# B&R Automation Studio project MIG1 (part 9)

### WSI_lib.c
```c
/********************************************************************
 * COPYRIGHT --
 ********************************************************************
 * Package: Lib
 * File: WSI_lib.c
 * Author: ckaczkowski
 * Created: June 18, 2014
 *******************************************************************/

#include <bur/plctypes.h>
#ifdef _DEFAULT_INCLUDES
	#include <AsDefault.h>
#endif

#ifndef _WSITYPES_C
#define _WSITYPES_C

//#define NULL 0

/* Prototyping of functions and function blocks */

float Scal(float x, AzzScal_typ* scale);
float LimScal(float x, AzzLimScal_typ* scale);

DINT Errors(ERROR_Mgr_typ *mgr , char type , unsigned short indx , unsigned long val);

DINT AckAllErrors(ERROR_Mgr_typ *mgr);

DINT StateVectorSrv(StateVectorProxy_typ *vect , UINT thread);

UINT Bool2Uint(plcbit in);
plcbit Uint2Bool(UINT in);

char* UDINT2ASC(UDINT val);
UDINT ASC2UDINT(char *p);

INT ABS_INT(INT x);

float getFromCalib(float x , Calib_Param_typ* calib , UINT type);

static UDINT hash_of_binary_array(char *key, int len);

///////////////////////////////////////////////////////
//////   Functions from Paul
void AzzLinSpline(AzzLinSpline_typ *lcr);
void AzzSlimPID(AzzSlimPID_typ *lcr);
void AzzRamp(AzzRamp_typ *lcr);
void AzzMovAvgFlt(AzzMovAvgFlt_typ *lcr) ;
void AzzLimScal(AzzLimScal_typ *lcr);
void AzzScal(AzzScal_typ *lcr);
void AzzTON(AzzTON_typ *t);
void HCRSPFazz(HCRSPFazz_type* inst);

void AzzLinSpline(AzzLinSpline_typ *lcr){
UINT outer , inner;
INT i;
float tempX, tempY;
float slope , delta;

	if(!lcr->pNodeVec)
		return;

	if(lcr->NbNodes < 2)
		return;

	//////////////////////////////////////////////

	if(lcr->Invert){

		if(lcr->x < lcr->pNodeVec[0].Y)
			lcr->y = lcr->pNodeVec[0].X;
		else if(lcr->x > lcr->pNodeVec[lcr->NbNodes-1].Y)
			lcr->y = lcr->pNodeVec[lcr->NbNodes-1].X;

		else{

			i = lcr->NbNodes-2;
			while((lcr->x < lcr->pNodeVec[i].Y) && (i > 0) ) { i--; }

			lcr->_i = i;

			delta = lcr->pNodeVec[i+1].Y - lcr->pNodeVec[i].Y;

			if(delta != 0.0)
				slope = (lcr->pNodeVec[i+1].X - lcr->pNodeVec[i].X)/delta;
			else
				slope =0;

			lcr->y = lcr->pNodeVec[i].X + slope * (lcr->x - lcr->pNodeVec[i].Y);

		}

	}
	else{

		if(lcr->x < lcr->pNodeVec[0].X)
			lcr->y = lcr->pNodeVec[0].Y;
		else if(lcr->x > lcr->pNodeVec[lcr->NbNodes-1].X)
			lcr->y = lcr->pNodeVec[lcr->NbNodes-1].Y;

		else{

			i = lcr->NbNodes-2;
			while((lcr->x < lcr->pNodeVec[i].X) && (i > 0) ) { i--; }

			lcr->_i = i;

			delta = lcr->pNodeVec[i+1].X - lcr->pNodeVec[i].X;

			if(delta != 0.0)
				slope = (lcr->pNodeVec[i+1].Y - lcr->pNodeVec[i].Y)/delta;
			else
				slope =0;

			lcr->y = lcr->pNodeVec[i].Y + slope * (lcr->x - lcr->pNodeVec[i].X);

		}

	}

	///////////////////////////////////////////////
	if(lcr->Update){
		lcr->Update = 0;

		//Bubble sort
		 for(outer=0;outer<lcr->NbNodes-1;outer++)
		 {
			 for(inner=outer+1;inner<lcr->NbNodes;inner++)
			 {

			 	if(lcr->Invert){

					 if(lcr->pNodeVec[outer].Y > lcr->pNodeVec[inner].Y)
					 {
						 tempX=lcr->pNodeVec[outer].X;
						 tempY=lcr->pNodeVec[outer].Y;

						 lcr->pNodeVec[outer].X = lcr->pNodeVec[inner].X;
						 lcr->pNodeVec[outer].Y = lcr->pNodeVec[inner].Y;

						 lcr->pNodeVec[inner].X = tempX;
						 lcr->pNodeVec[inner].Y = tempX;

					 }

			 	}
				else{

					if(lcr->pNodeVec[outer].X > lcr->pNodeVec[inner].X)
					 {
						 tempX=lcr->pNodeVec[outer].X;
						 tempY=lcr->pNodeVec[outer].Y;

						 lcr->pNodeVec[outer].X = lcr->pNodeVec[inner].X;
						 lcr->pNodeVec[outer].Y = lcr->pNodeVec[inner].Y;

						 lcr->pNodeVec[inner].X = tempX;
						 lcr->pNodeVec[inner].Y = tempX;

					 }

				}
			 }
		 }

	}

}

void AzzTON(AzzTON_typ *t) {
  if (t->IN) {
    // Check for rising edge
    if (!t->M) {
      t->StartTime = clock_ms();
    }

    // Determine elapsed time
    t->ET = clock_ms() - t->StartTime;

    // Check if the elapsed time has reached delay time
    if (t->ET >= t->PT) {
      t->Q = 1;
      t->ET = t->PT;
    } else {
      t->Q = 0;
    }

  } else {
    t->Q = 0;
    t->ET = 0;
  }

  // Set M to IN to allow checking for rising edge
  t->M = t->IN;
}

void AzzRamp(AzzRamp_typ *lcr) {
float x = lcr->x, y = lcr->y_old;
float dt;
DINT time , deltaT;

	lcr->status = 0;

	if ( !lcr->enable ) {

		lcr->timestore1 = AsIOTimeStamp();
		lcr->status = 65534;
		return;

	}

	// Check parameters
	  // rate up and rate down have to be greater than zero
	if ( lcr->dy_up <= 0 || lcr->dy_down <= 0 ) {
	  lcr->status = 12034;
	  return;
	}

	if ( lcr->set ) { // Set default value

		lcr->set = 0;

		y = lcr->y_set;

		lcr->y_old = y;

		lcr->y = y;

		lcr->timestore1 = AsIOTimeStamp();

	}
	else {
		// Process Ramp

		time = AsIOTimeStamp();
		deltaT = (time- lcr->timestore1);
		lcr->timestore1 = time;

		if(deltaT > 0 && (deltaT < 0x4FFFFFFF))
			dt = (float)(deltaT) / 1000000.0;
		else
			dt = 0.0;

		lcr->dt = dt;

		/*
		// Calculate new value
		if ( x > y && y > 0 ) {
			y = lcr->y_old + ( dt * lcr->dy_up );
			if(y > x)
				y = x;

		} else if ( x < y && y < 0 ) {
			y = lcr->y_old - ( dt * lcr->dy_up );
			if(y < x)
				y = x;

		} else if ( x < y && y > 0 ) {
			y = lcr->y_old - ( dt * lcr->dy_down );
			if(y < x)
				y = x;

		} else if ( x > y && y < 0 ) {
			y = lcr->y_old + ( dt * lcr->dy_down );
			if(y > x)
				y = x;
		}
		*/

		if ( x > y ) {
			y = lcr->y_old + ( dt * lcr->dy_up );
			if(y > x)
				y = x;

		} else if ( x < y ) {
			y = lcr->y_old - ( dt * lcr->dy_down );
			if(y < x)
				y = x;
		}

		// Check limits
		if (y >= lcr->y_max ) {
		  y = lcr->y_max;
		  lcr->max_limit = 1;

		}

		else if(y <= lcr->y_min ) {
		  y = lcr->y_min;
		  lcr->min_limit = 1;

		}

		lcr->y = y;

		lcr->x_reached = (lcr->y == lcr->x)? 1:0;
		lcr->y_old = y;

	}

}

void AzzMovAvgFlt(AzzMovAvgFlt_typ *lcr) {

  float *ptr;
  double *sum = (double*)&lcr->sum_old;
  int i;

  //lcr->y = lcr->x ;
  //return;

  if(!lcr){
  	lcr->status = -1;
	return;
  }

  if(lcr->base == 0){
  	lcr->status = -2;
	return;
  }

  lcr->status = 0;

  if ( lcr->enable ) {
    // Default to successful status
    lcr->status = 0;

    // If base has changed, re-allocate buffer
    if ( lcr->base != lcr->base_old || ( (void *)lcr->p_xold == 0 ) ) {

      // Free the old buffer
	 if((lcr->p_xold != 0 ) && lcr->base_old > 0){
		  if(TMP_free(lcr->base_old , (void**) lcr->p_xold)){
		  	return;
		  }
		  else
		  	lcr->base_old = 0;

	 }
	 else{ // Memory leack

	 	 lcr->base_old = 0;
		 lcr->p_xold = 0;

	 }

      //if ( (void *)lcr->p_xold != 0 )
        //free((void *)lcr->p_xold);

      // Allocate new buffer
      //lcr->p_xold = (unsigned long)malloc(lcr->base * sizeof(lcr->x));
      if(TMP_alloc(lcr->base * sizeof(float)  , (void**)&lcr->p_xold))
	  	return;
	  else
		lcr->base_old = lcr->base;

      ptr = (float*)lcr->p_xold;

      // Set buffer to initial values (current x)
      if (ptr != 0) {
        // Loop through whole buffer
        for( i = 0; i < lcr->base; i++ ) {
          *ptr = lcr->x;
          ptr++;
        }
      } else {
        lcr->status = 12018;
        return;
      }

      // Set sum
      *sum = lcr->x * lcr->base;

	  lcr->y = (*sum) / lcr->base;

      // Set index
      lcr->i_xold = 0;
    }

	 //return;
	if ( lcr->i_xold >= lcr->base )
      lcr->i_xold = 0;

	ptr = (float*)lcr->p_xold;
    // Calculate new sum
    *sum = *sum - *(ptr + lcr->i_xold) + lcr->x;

    // Replace x value in buffer
    *(ptr + lcr->i_xold) = lcr->x;

    // Increase index and ring around the buffer if necessary
    lcr->i_xold ++;

    // Calculate new avg
    lcr->y = (*sum) / lcr->base;

  }

  else {

    lcr->status = 65534;
  }

}

void AzzSlimPID(AzzSlimPID_typ *lcr) {

  AzzPID_typ *pid = &lcr->PID_inst;
  azzslimpid_par_typ *para = lcr->pPar;
  float p, i, d, error, dt;
  DINT time , deltaT;

  // TODO - Ensure that the derivative term does not go crazy first scan
  // We are not using the derivative

  if (lcr->enable) {
	    // Get current time
	    time = AsIOTimeStamp();

	    // Determine error
	      // Includes feedback damping
	      // e_fbk = Kfbk / Kp * (Ytotal - Y)

	    //error = lcr->W - lcr->X - pid->e_fbk;
	    error = lcr->W - lcr->X ;

		deltaT = (time - pid->last_time);

		if(deltaT > 0 && (deltaT < 0x4FFFFFFF))
	    	dt = (float)(deltaT) / 1000000.0;
		else
			dt = 0.0;

		lcr->dt = dt;
		lcr->e = error;

	    // Proportional control
	    p = para->Kp * error;

	    // Integral control
	    //pid->i_sum += error * dt;
	    pid->i_sum += ((error - pid->e_fbk) * para->Kp * dt);

		if(para->Tn > 0)
	    	i = pid->i_sum / para->Tn;
		else
			i = 0;

	    // Derivative control
	    if(dt > 0)
	    	d = ((lcr->X - pid->d_old) / dt) * para->Tv * para->Kp ;
		else
			d = 0.0;

	    pid->d_old = lcr->X;

	    // Set output variable
	    lcr->Y = p + i + d;

	    // Limit output variable
	    if (lcr->Y > para->Y_max) {
	      pid->e_fbk = para->Kfbk * (lcr->Y - para->Y_max);
	      lcr->Y = para->Y_max;
	    } else if (lcr->Y < para->Y_min) {
	      pid->e_fbk = para->Kfbk * (lcr->Y - para->Y_min);
	      lcr->Y = para->Y_min;
	    } else {
	      pid->e_fbk = 0;
	    }

  } else {

  	i = pid->i_sum = 0;
    lcr->status = 65534;
  }

  pid->last_time = AsIOTimeStamp();

}

void AzzScal(AzzScal_typ *lcr) {
  REAL k, d;

  if (lcr->x1 != lcr->x2) {
    k = (lcr->y2 - lcr->y1) / (lcr->x2 - lcr->x1);
    lcr->y = lcr->y1 + (k * (lcr->x - lcr->x1));

  } else {
    lcr->y = 0;
  }

}

void AzzLimScal(AzzLimScal_typ *lcr) {
  REAL *high, *low;

  // Run LCRScal - this function is the same except for limits
  AzzScal((AzzScal_typ *)lcr);

  // Find high limit and low limit
  if (lcr->y1 < lcr->y2) {
    high = &lcr->y2;
    low = &lcr->y1;
  } else {
    low = &lcr->y2;
    high = &lcr->y1;
  }

  // Limit y to be between the high and low values
  if (lcr->y > *high)
    lcr->y = *high;
  if (lcr->y < *low)
    lcr->y = *low;

}

//////////    END of New Functions /////////////////////
/////////////////////////////////////////////////////

float LimScal(float x, AzzLimScal_typ* scale){

	scale->x = x;
	AzzLimScal(scale);

	return scale->y;
}

float Scal(float x, AzzScal_typ* scale){

	scale->x = x;
	AzzScal(scale);

	return scale->y;
}

DINT Errors(ERROR_Mgr_typ *mgr , char type , unsigned short indx , unsigned long val){

	if(!mgr->logs[indx].status){

		mgr->lastItemIndx++;
		if(mgr->lastItemIndx >= 64)
			mgr->lastItemIndx = 0;

		mgr->logs[indx].status = 1;
		mgr->logs[indx].value = val;
		mgr->history[mgr->lastItemIndx] = indx;

		if(type > 0){
			if(type >= mgr->Error) // set only higher priority error
				mgr->Error = type;
		}
		else
			mgr->Error = type;

		return 1;

	}
	else
		return 0;
}

DINT AckAllErrors(ERROR_Mgr_typ *mgr){
	int i;

	// Never clear fatal error
	if (mgr->Error < 0)
		return -1;

	for( i = 0 ; i < 64 ; i++){

		mgr->logs[i].status = 0;

		mgr->history[i] = 0;

	}

	mgr->Error = 0;
	mgr->lastItemIndx = 0;

	return 1;

}

DINT StateVectorSrv(StateVectorProxy_typ *vect , UINT thread){

	if(vect->testMode)
		return;

	/*****************************************/
	///    VECTOR  SERVER

	if(!vect->simul){

		vect->OutVect.Mode = vect->Mode ;

		switch(vect->Mode){

			case vectSt_Mode_Idle:

				vect->OutVect.volt = 0.0;
				vect->OutVect.vel = 0.0;

				break;

			case vectSt_Mode_Hold:

				break;

			case vectSt_Mode_Home:

				break;

			case vectSt_Mode_Pos:

				vect->OutVect.volt = 0.0;
				vect->OutVect.amp  = 0.0;

				//if(thread == vect->Indx )
					vect->OutVect.x = vect->InVal;

				break;

			case vectSt_Mode_Vel:

				vect->OutVect.volt = 0.0;
				vect->OutVect.amp  = 0.0;

				//if(thread == vect->Indx )
					vect->OutVect.vel = vect->InVal;

				break;

			case vectSt_Mode_Volt:

				vect->OutVect.amp  = 0.0;

				//if(thread == vect->Indx )
					vect->OutVect.volt = vect->InVal;

				vect->OutVect.vel = 0;

				break;

			case vectSt_Mode_Torq:

				vect->OutVect.volt = 0.0;

				//if(thread == vect->Indx )
					vect->OutVect.amp = vect->InVal;

				vect->OutVect.vel = 0;

				break;

			case vectSt_Mode_PT:

				vect->OutVect.volt = 0.0;
				vect->OutVect.amp  = 0.0;
				vect->OutVect.x = vect->InVal;

				break;

		}
	}
	else{

		vect->FbkVect.Mode = vect->Mode;

		switch(vect->Mode){

			case vectSt_Mode_Idle:

				vect->FbkVect.x = 0;
				vect->FbkVect.vel = 0;

				break;

			case vectSt_Mode_Hold:

				break;

			case vectSt_Mode_Home:

				break;

			case vectSt_Mode_Pos:

				vect->FbkVect.x = vect->InVal;

				break;

			case vectSt_Mode_Vel:

				vect->FbkVect.vel = vect->InVal;

				break;

			case vectSt_Mode_Volt:

				vect->FbkVect.volt = vect->InVal;

				break;

			case vectSt_Mode_Torq:

				vect->FbkVect.amp = vect->InVal;

				break;

			case vectSt_Mode_PT:

				vect->FbkVect.x = vect->InVal;
				//vect->OutVect.x = vect->InVal;

				break;

		}

	}

	return 1;

}

UINT Bool2Uint(plcbit in){

	if(in)
		return 1;
	else
		return 0;

}

plcbit Uint2Bool(UINT in){

	if(in > 0)
		return 1;
	else
		return 0;

}

char* UDINT2ASC(UDINT val){
static char ret[5];
UDINT mask;
int i;

	mask = 0x000000FF;

	for(i=3 ; i >= 0 ; i--){

		ret[i] = (char)(val & mask);
		val = val >> 8;

	}
	ret[4] = 0;
	return ret;

}

UDINT ASC2UDINT(char *p){
UDINT val;
int i;

	val = 0;

	for(i=0 ; i < 4  ; i++){
		val = val<<8;
		val += p[i];
	}

	return val;

}
INT ABS_INT(INT x){

	if( x >= 0)
		return x;
	else
		return x*(-1);

}

float getFromCalib(float x , Calib_Param_typ* calib , UINT type){
float ret; float _x;
AzzScal_typ scale;

	if(!calib)
		return 0.0;

	if(x == 0.0)
		return 0.0;

	if(x < 0.0)
		_x = x * (-1.0);
	else
		_x = x;

	switch(type){

		case CALIB_ONE2ONE:

			ret = _x;

		break;

		case CALIB_2POINTS:

			scale.x = _x;
			scale.x1 = calib->val[0];
			scale.y1 = calib->val[1];
			scale.x2 = calib->val[2];
			scale.y2 = calib->val[3];

			if( _x < scale.x1)
				ret = (_x/scale.x1) * scale.y1;

			else {
				AzzScal(&scale);
				ret = scale.y;
			}

		break;

		case CALIB_2POINTS_4OFF:

			scale.x = _x;
			scale.x1 = calib->val[4];
			scale.y1 = calib->val[5];
			scale.x2 = calib->val[6];
			scale.y2 = calib->val[7];

			if( _x < scale.x1)
				ret = (_x/scale.x1) * scale.y1;

			else {
				AzzScal(&scale);
				ret = scale.y;
			}

		break;

		case CALIB_2POINTS_INV:

			scale.x = _x;
			scale.x1 = calib->val[1];
			scale.y1 = calib->val[0];
			scale.x2 = calib->val[3];
			scale.y2 = calib->val[2];

			if( _x < scale.x1)
				ret = (_x/scale.x1) * scale.y1;

			else {
				AzzScal(&scale);
				ret = scale.y;
			}

		break;

		case CALIB_2POINTS_4OFF_INV:

			scale.x = _x;
			scale.x1 = calib->val[5];
			scale.y1 = calib->val[4];
			scale.x2 = calib->val[7];
			scale.y2 = calib->val[6];

			if( _x < scale.x1)
				ret = (_x/scale.x1) * scale.y1;

			else {

				AzzScal(&scale);
				ret = scale.y;
			}

		break;

	}

	// Symetric to zero
	if(x <  0.0)
		ret = ret * (-1.);

	return ret;

}

static UDINT hash_of_binary_array(char *key, int len)
{
	unsigned int hash, i;
	for(hash = i = 0; i < len; ++i)
	{
		hash += key[i];
		hash += (hash << 10);
		hash ^= (hash >> 6);
	}
	hash += (hash << 3);
	hash ^= (hash >> 11);
	hash += (hash << 15);
	return hash;
}

///   New Path Generator created March 2019 by CK
void HCRSPFazz(HCRSPFazz_type* inst){
float dist, a , d , v , v02 , ad2 , x , s ;
float S_end , S_in , V_in , V0 , V_max;
float dir;
UINT t;
float deltaT;

	if(!inst)
		return;
/*****************************************/

	if(!inst->Intr._Set_home && inst->Set_home){
		// This is new for conveniance
		inst->Set_home = 0;

		inst->s_set = inst->s_home;
		inst->v_set = 0;
		inst->a_set = 0;

		inst->Intr.step = 0;

	}

	if(!inst->Intr._Stop && inst->Stop){

		// This is new for conveniance
		inst->Stop = 0;

		inst->v_set = 0;
		inst->a_set = 0;

		inst->Intr.step = 0;

	}

	if(!inst->Intr._Brake && inst->Brake){

		d = (inst->v_set > 0)? inst->pMove_Para->aDec_pos : inst->pMove_Para->aDec_neg;
		dir = (inst->v_set > 0.0)? 1.0:-1.0;

		/*
		inst->s_end = ((inst->v_set * inst->v_set )/d/2.0)*dir + inst->s_set;

		inst->Intr.step = 1;
		*/

		inst->Intr.S0 = ((inst->v_set * inst->v_set )/d/2.0)*dir;
		inst->Intr.segm[0].s = inst->Intr.S0  + inst->s_set ;
		inst->Intr.segm[0].v = 0;
		inst->Intr.segm[0].a = -d * dir;

		inst->Intr.S1 = 0.0;
		inst->Intr.segm[1].s = inst->Intr.segm[0].s;
		inst->Intr.segm[1].v = 0;
		inst->Intr.segm[1].a = 0;

		inst->Intr.S2 = 0.0;
		inst->Intr.segm[2].s = inst->Intr.segm[0].s;
		inst->Intr.segm[2].v = 0;
		inst->Intr.segm[2].a = 0;

		inst->Intr.S3 = 0.0;
		inst->Intr.segm[3].s = inst->Intr.segm[0].s;
		inst->Intr.segm[3].v = 0;
		inst->Intr.segm[3].a = 0;

		inst->Intr.indx = 0;
		inst->elapseTime = 0.0;
		inst->Reached = 0;
		inst->Intr.step = 3;

	}

	if(!inst->Intr._Init && inst->Init )
		inst->Intr.step = 1;

	switch(inst->Intr.step){

		//// Verify if current velocity in bigger then maximum velocity
		case 1:

			strcpy(inst->Intr.statusTxt , "");

			inst->Reached = 0;

			inst->Intr.segm[0].s = inst->s_set;
			inst->Intr.segm[0].v = inst->v_set;
			inst->Intr.segm[0].a = 0.0;

			inst->Intr.S0 = 0;
			////////////////////////////////////////////////////////////////////////////////////////
			// Check if movement direction change is necessary

			dist = inst->s_end - inst->Intr.segm[0].s;
			d = (inst->Intr.segm[0].v > 0)? inst->pMove_Para->aDec_pos : inst->pMove_Para->aDec_neg;

			s = ((inst->v_set * inst->v_set)/d)/2.0;

			if((fabsf(dist) < s) 					// Distance is smaller then coming from deceleration
				|| ((dist *  inst->v_set)<0.0)){ 	// Running in oposite direction

				strcpy(inst->Intr.statusTxt , "Change move direction");

				if(inst->Intr.segm[0].v > 0){

					inst->Intr.S0 = s;
					inst->Intr.segm[0].s += s;
					inst->Intr.segm[0].v = 0.0;
					inst->Intr.segm[0].a = -d;

				}
				if(inst->Intr.segm[0].v < 0){

					inst->Intr.S0 = -s;
					inst->Intr.segm[0].s -= s;
					inst->Intr.segm[0].v = 0.0;
					inst->Intr.segm[0].a = d;

				}

				goto CALCULATE_TRAPEZOID;

			}

			///////////////////////////////////////////////////////////////////////////////////////////
			///  Check Speed above maximum

			if(inst->v_set > 0.0)
				V_max = inst->pMove_Para->vC_pos;
			else if(inst->v_set < 0.0)
				V_max = inst->pMove_Para->vC_neg;

			if(fabsf(inst->v_set) > V_max){ // reduce speed first{

				if(inst->v_set > 0.0){

					inst->Intr.segm[0].v = V_max;
					inst->Intr.segm[0].a = -inst->pMove_Para->aDec_pos;

					x = (fabsf(inst->v_set) - V_max );
					inst->Intr.S0 = (x * x)/ inst->pMove_Para->aDec_pos /2.0 ;
					inst->Intr.S0 += inst->Intr.segm[0].v * x/inst->pMove_Para->aDec_pos;

					inst->Intr.segm[0].s += inst->Intr.S0;

					strcpy(inst->Intr.statusTxt , "Max Pos Vel");
				}
				else if(inst->v_set < 0.0){

					inst->Intr.segm[0].v = -V_max;
					inst->Intr.segm[0].a = inst->pMove_Para->aDec_neg;

					x = (fabsf(inst->v_set) - V_max );
					inst->Intr.S0 = (x * x)/ inst->pMove_Para->aDec_neg /(-2.0) ;
					inst->Intr.S0 += inst->Intr.segm[0].v * x/inst->pMove_Para->aDec_neg;

					inst->Intr.segm[0].s += inst->Intr.S0;

					strcpy(inst->Intr.statusTxt , "Max Neg Vel");
				}

			}

			CALCULATE_TRAPEZOID:
			//////////////////////////////////////////////////////////
			///  Calculate Segments 1 , 2 , 3
			S_end = inst->s_end;
			S_in  = inst->Intr.segm[0].s ;
			V_in  = inst->Intr.segm[0].v ;

			dir = (S_end > S_in)? 1.0:-1.0;

			if(dir > 0){
				a = inst->pMove_Para->aAcc_pos;
				d = inst->pMove_Para->aDec_pos;
			}
			else if(dir < 0){

				a = inst->pMove_Para->aAcc_neg;
				d = inst->pMove_Para->aDec_neg;
			}
			else{

				strcpy(inst->Intr.statusTxt , "No Trapezoid");

			}

			inst->Intr.segm[1].a = a ;
			inst->Intr.segm[2].a = 0;
			inst->Intr.segm[3].a = -d  ;

			////////////////////////////////////////////
			// Calculate maximum velocity

			dist = fabsf(S_end - S_in);
			V0 = fabsf(V_in);

			v02 = (V0 * V0)/ (2.0 * a);
			ad2 = (1.0/(2*a)) + (1.0/(2*d));

			 v = (dist + v02)/ad2;

			 v = sqrtf(v);

			////////////////////////

			if(dir > 0.0){	 // positive move direction

				if(v > inst->pMove_Para->vC_pos){

					inst->Intr.segm[1].v = inst->pMove_Para->vC_pos;
				}
				else{

					inst->Intr.segm[1].v = v;

				}
			}

			else if(dir < 0.0){	 // negative move direction

				if( v > inst->pMove_Para->vC_neg){

					inst->Intr.segm[1].v = inst->pMove_Para->vC_neg ;
				}
				else{

					inst->Intr.segm[1].v = v ;

				}
			}

			inst->Intr.segm[2].v = inst->Intr.segm[1].v;
			inst->Intr.segm[3].v = 0.0;

			////////////////////////////////////

			inst->Intr.S1 = 0.0; // Init with 0

			x = inst->Intr.segm[1].v - V0;
			x = x*x;
			x = x/(2.0 * a);

			inst->Intr.S1 += x; // + Triangle area

			///

			x = V0 * (inst->Intr.segm[1].v - V0);
			x = x /(2.0 * a) ;

			inst->Intr.S1 += x; // + Square area
			inst->Intr.S1 = inst->Intr.S1 * dir;
			inst->Intr.segm[1].s = inst->Intr.S1 + inst->Intr.segm[0].s ;

			//////////////////////////////

			inst->Intr.S3 = (inst->Intr.segm[2].v *  inst->Intr.segm[2].v)/( 2*d)* dir ; // Area under deceleration
			inst->Intr.S2 = (S_end - S_in) - inst->Intr.S1 - inst->Intr.S3;

			inst->Intr.segm[2].s = S_end - inst->Intr.S3;
			inst->Intr.segm[3].s = S_end;

			inst->Intr.segm[1].v = inst->Intr.segm[1].v * dir ;
			inst->Intr.segm[2].v = inst->Intr.segm[2].v * dir ;
			inst->Intr.segm[3].v = inst->Intr.segm[3].v * dir ;

			inst->Intr.segm[1].a = inst->Intr.segm[1].a * dir ;
			inst->Intr.segm[2].a = 0;
			inst->Intr.segm[3].a = inst->Intr.segm[3].a * dir ;

			inst->ApproachDir =(inst->Intr.segm[2].v > 0)? 1:-1;
			if(inst->Intr.segm[2].v == 0)
				inst->ApproachDir = 0;

			/////////////////////////////
			inst->Intr.indx = 0;
			inst->elapseTime = 0.0;

			// This is new for conveniance
			inst->Init = 0;

			//inst->Intr.step++;
			//inst->Intr.step++;
			inst->Intr.step = 3;

		break;

		case 3:

			inst->Reached = 0;

			if(inst->Intr.TaskPeriod <= 0.0)
				inst->Intr.TaskPeriod = 0.0024; // standard time

			inst->elapseTime += inst->Intr.TaskPeriod;

			inst->a_set = inst->Intr.segm[inst->Intr.indx].a;
			inst->v_set = inst->Intr._v_set +  inst->Intr.segm[inst->Intr.indx].a * inst->Intr.TaskPeriod;
			inst->s_set = inst->Intr._s_set +  (inst->v_set + inst->Intr._v_set)/2.0 * inst->Intr.TaskPeriod;

			if((inst->s_set > inst->Intr._s_set)){

				if(inst->s_set >= inst->Intr.segm[inst->Intr.indx].s){

					inst->v_set = inst->Intr.segm[inst->Intr.indx].v;
					inst->Intr.indx++;

				}
			}

			else if((inst->s_set < inst->Intr._s_set)){

				if(inst->s_set <= inst->Intr.segm[inst->Intr.indx].s){

					inst->v_set = inst->Intr.segm[inst->Intr.indx].v;
					inst->Intr.indx++;

				}
			}

			else if (fabsf(inst->s_set - inst->Intr.segm[inst->Intr.indx].s) < 0.01) {

				strcpy(inst->Intr.statusTxt , "END END");

				inst->s_set = inst->Intr.segm[inst->Intr.indx].s;
				inst->v_set = inst->Intr.segm[inst->Intr.indx].v;
				inst->Intr.indx++;

			}

			if(inst->Intr.indx > 3){

				inst->s_set = inst->Intr.segm[3].s;
				inst->v_set = inst->Intr.segm[3].v;
				inst->a_set = 0.0;

				inst->Reached = 1;

				// This is new for conveniance
				inst->Brake = 0;

				inst->Intr.step = 0;

			}

		break;

		default:

			strcpy(inst->Intr.statusTxt , "Idle");

			inst->Intr.step = 0;

		break;

	}

	inst->MoveDir =(inst->v_set > 0)? 1:-1;
	if(inst->v_set == 0.0)
		inst->MoveDir = 0;

/****************************************/
	inst->Intr._s_set = inst->s_set ;
	inst->Intr._v_set = inst->v_set ;
	inst->Intr._a_set = inst->a_set ;

	inst->Intr._enable = inst->enable ;
	inst->Intr._Stop = inst->Stop ;
	inst->Intr._Set_home = inst->Set_home ;
	inst->Intr._Init = inst->Init ;
	inst->Intr._Brake = inst->Brake ;

}

#endif
```

### WSI_types.h
```c
/********************************************************************
 * COPYRIGHT -- wsi
 ********************************************************************
 * Package:
 * File: WSI_types.h
 * Author: ckaczkowski
 * Created: 17 June 2014
 *******************************************************************/

#include <bur/plctypes.h>

#ifndef _WSITYPES_H
#define _WSITYPES_H

#include <..\lib\Statelib.h>
//#include <..\Universal\SuperDefinition.h>

#if 0
#define PARAM_NUM_MAX  		256
#define PARAM_INT_NUM_MAX  	8
#define PARAM_ENUM_NUM_MAX  32
#define PARAM_STR_NUM_MAX   16
//#define PARAM_ENUM_NUM_MAX  8
//#define PARAM_STR_NUM_MAX   8
#define VAR_NUM_MAX    		128
#define ENUM_VAR_MAX   		32
#define INT_VAR_MAX    		32
#define STR_VAR_MAX    		64
//#define SEGM_NUM_MAX   		31
#define SEGM_NUM_MAX   		32
#define TXT_RESOURCES_MAX 	64
#define RES_TXT_LEN 		16
#define PAGES_MAX			64

#endif

#define CALIB_ONE2ONE			0
#define CALIB_2POINTS 			1
#define CALIB_2POINTS_4OFF 		2
#define CALIB_2POINTS_INV 		3
#define CALIB_2POINTS_4OFF_INV	4

#define CALC_SLOPE_BOTH			10

/////////////////////////////////////////////////////
typedef struct AzzNode_typ
{
	float X;
	float Y;

} AzzNode_typ;

typedef struct AzzLinSpline
{
	/* VAR_INPUT (analog) */
	unsigned short NbNodes;
	AzzNode_typ* pNodeVec;
	unsigned char Smooth;
	float Rness;
	signed char DisMode;
	float x;
	/* VAR_OUTPUT (analog) */
	float y;
	unsigned short status;
	/* VAR (analog) */
	INT _i;
	/* VAR_INPUT (digital) */
	plcbit enable;
	plcbit Invert;
	plcbit Update;
} AzzLinSpline_typ;

// New Functions from Paul
typedef struct AzzTON {
  BOOL IN;
  TIME PT;
  BOOL Q;
  TIME ET;
  TIME StartTime;
  BOOL M;
  UDINT Restart;
} AzzTON_typ;

typedef struct AzzMovAvgFlt {
	/* VAR_INPUT (analog) */
	float x;
	unsigned long base;
	/* VAR_OUTPUT (analog) */
	unsigned short status;
	float y;
	/* VAR (analog) */
	double sum_old;
	//signed long sum_old_dbl_2;
	unsigned long p_xold;
	unsigned short i_xold;
	unsigned long base_old;
	unsigned long bootkey_old;
	/* VAR_INPUT (digital) */
	plcbit enable;
	/* VAR (digital) */
	plcbit enable_old;
} AzzMovAvgFlt_typ;

typedef struct AzzPIDTune{
	float nothing;

} AzzPIDTune_typ;

typedef struct AzzPID{
	float i_sum, d_old, e_fbk;
	DINT last_time;
} AzzPID_typ;

typedef struct azzslimpid_par {
	float Y_max;
	float Y_min;
	float Kp;
	float Tn;
	float Tv;
	float Kfbk;
} azzslimpid_par_typ;

typedef struct AzzSlimPID{
	/* VAR_INPUT (analog) */
	float W;
	float X;
	unsigned long request;
	azzslimpid_par_typ* pPar;
	/* VAR_OUTPUT (analog) */
	float e;
	float Y;
	float dt;
	unsigned short status;
	unsigned short addInfo;
	/* VAR (analog) */
	AzzMovAvgFlt_typ MovAvgFlt_inst;
	AzzPIDTune_typ PIDTune_inst;
	AzzPID_typ PID_inst;
	unsigned long requ_old;
	/* VAR_INPUT (digital) */
	plcbit enable;
	/* VAR (digital) */
	plcbit enable_old;
} AzzSlimPID_typ;

typedef struct AzzRamp{
	/* VAR_INPUT (analog) */
	float x;
	float dy_up;
	float dy_down;
	float y_max;
	float y_min;
	float y_set;
	/* VAR_OUTPUT (analog) */
	unsigned short status;
	float y;
	/* VAR (analog) */
	float dt;
  	float y_old;
	//signed long y_dbl_1;
	//signed long y_dbl_2;
	unsigned long timestore1;
	//unsigned long timestore2;
	//unsigned long getDtForceOff;
	//struct SysInfo sysinfo_inst;
	/* VAR_INPUT (digital) */
	plcbit enable;
	plcbit set;
	/* VAR_OUTPUT (digital) */
	plcbit x_reached;
	plcbit max_limit;
	plcbit min_limit;
} AzzRamp_typ;

typedef struct AzzLimScal {
  REAL x, x1, y1, x2, y2, y;
} AzzLimScal_typ;

typedef struct AzzScal{
  REAL x, x1, y1, x2, y2, y;
} AzzScal_typ;

//////////////////////////////////////////
///////////////////////////////////////////////////////////

typedef struct LogItem_typ{

	signed long timeStamp;
	signed short status;
	unsigned long value;
	plcstring  txt[32];

}LogItem_typ;

typedef struct WarnItem_typ{
	signed short status;
	plcstring  txt[32];

}WarnItem_typ;

typedef struct ERROR_Mgr_typ{
	SINT Error;
	unsigned short lastItemIndx;
	unsigned short history[128];
	LogItem_typ logs[128];
	UINT warnings;

}ERROR_Mgr_typ;

/*********************************************************************/

/***********   VECTOR STATE        ***************************************/

/*********************************************************************/

#define vectSt_Mode_OFF 0
#define vectSt_Mode_Idle 1
#define vectSt_Mode_Hold 2
#define vectSt_Mode_Home 3
#define vectSt_Mode_Pos 4
#define vectSt_Mode_Vel 5
#define vectSt_Mode_Torq 6
#define vectSt_Mode_Volt 7
#define vectSt_Mode_PT 	 8
#define vectSt_Move_Abs  9
#define vectSt_Move_Rel  10
#define vectSt_Mode_Custom 11
#define vectSt_Mode_Drive_Independant 12

/******   Generic Vector Command to TML *************/
#define VECT_UpdateSignFilter		1
#define VECT_ClearSignFilter		2
#define VECT_FullSignFilter			3
#define VECT_Set_Gain				4
#define VECT_Set_Gain_Zero			5
#define VECT_Set_PID_Param			6
#define VECT_Set_SATP				7
#define VECT_Set_SATP_Zero			8

#define VECT_Set_Param_0			10
#define VECT_Set_Param_1			11
#define VECT_Set_Param_2			12
#define VECT_Set_Param_3			13
#define VECT_Set_Param_4			14
#define VECT_Set_Param_5			15
#define VECT_Set_Param_6			16
#define VECT_Set_Param_7			17
#define VECT_Set_MaxError			18

#define VECT_Set_CmdWord			20

#define VECT_OSC_Start_Cmd			40
#define VECT_OSC_Stop_Cmd			41
#define VECT_OSC_Update_Cmd			42
#define VECT_OSC_Stop2_Cmd			43

#define VECT_Move_Abs_Cmd			22

#define VECT_Move_Rel_Cmd			23
#define VECT_Move_Stop_Cmd			24

#define VECT_ARC_Stop_Cmd			25
#define VECT_ARC_Start_Cmd			26

#define VECT_ZERO_AMPS_Cmd			27
#define VECT_DEFAULT_AMPS_Cmd		28

#define VECT_RESTART_SRV_Cmd		29

#define VECT_Set_KPP				30
#define VECT_Set_KPP_Zero			31

#define VECT_Upd_CACC				32
#define VECT_Upd_CSPD				33

#define VECT_Set_Act_Pos			35

#define VECT_Set_OUT0				50
#define VECT_Rst_OUT0				51
#define VECT_Set_OUT1				52
#define VECT_Rst_OUT1				53
#define VECT_Set_OUT2				54
#define VECT_Rst_OUT2				55
#define VECT_Set_OUT3				56
#define VECT_Rst_OUT3				57
#define VECT_Set_OUT4				58
#define VECT_Rst_OUT4				59

#define VECT_Set_FFL				60

#define VECT_Refresh_Mode			70

#define VECT_Set_OSC_Max 		80
#define VECT_Set_OSC_Min 		81
#define VECT_Set_OSC_Time		82
#define VECT_Set_OSC_DwellIn 	83
#define VECT_Set_OSC_DwellOut 	84
#define VECT_Set_OSC_Steer		85
#define VECT_Set_OSC_Cmd_Param 	86
#define VECT_Set_OSC_Jog_Volt	87
#define VECT_Set_OSC_Jog_Speed	88
#define VECT_Set_OSC_Jog_Step	89
#define VECT_Set_OSC_Amplit 	90
#define VECT_Set_OSC_AllParam 	91
#define VECT_Set_OSC_Home 		92
#define VECT_Set_All_Run_Param 	93

#define VECT_Set_CACC			100
#define VECT_Get_APOS			101
#define VECT_STOP				102
#define VECT_EINT				103

#define VECT_Cmd_SAP			110
#define VECT_Cmd_CPA			111
#define VECT_Cmd_CACC			112
#define VECT_Cmd_CPOS			113

#define VECT_Cmd_MIG_OSC		120

#define VECT_Read_MCR			130

#define VECT_UPD_Cmd			135
#define VECT_Move_Abs_Param		136

typedef struct STATE_VECTOR_typ
{
	//plcbit OK;
	float x; 	// value
	float x2; 	// value
	float vel; 	// first derivative
	float acc; 	// second derivative
	float amp; 	// current amps
	float volt; // volts
	float softLimits[2]; // software limits
	//DINT Center;
	float Center;
	signed short Status;
	signed short Mode;

}STATE_VECTOR_typ;

typedef struct StateVectorProxy_typ{
	plcstring Name[16];
	UINT Indx;
   /* VAR_INPUT (analog) */
   UINT simul;
   UINT testMode;
   UINT xCMD;
   UINT cmdWord;
   float fParam[8];
   DINT Param[8];
   unsigned short MCRReg;
   unsigned long StatusReg;
   USINT xCmd_busy;
   float InVal;
   float maxVel;
   float maxAcc;
   unsigned short curStep;
   signed short Mode;
   /* VAR_OUTPUT (analog) */
   STATE_VECTOR_typ OutVect;
   signed short Status;
   STATE_VECTOR_typ FbkVect;
   DINT actPosDINT;
   INT FbkWarning;
   UDINT VirStatus;

}StateVectorProxy_typ;

/******* Files Operation***************/

#define PRG_FILE_EXT ".prg"
#define PRG_NO_NEXT "None"

#define F_READ 				1
#define F_WRITE 			2
#define F_DELETE			3
#define F_FREE_MEM 			4

#define F_LOAD_CURCFG		5
#define F_SAVE_CURCFG		6
#define F_SAVE_AS_CURCFG	7

#define F_RENAME			8
#define F_COPY				9
#define F_GET_NEXT_FILE		10
#define F_SET_NEXT_FILE		11
#define F_READ_FILE_TO_TMP 	12
#define F_SAVE_AS_TMP 		13

#define F_READ_DIR 			20
#define F_READ_FILE_INF 	21
#define F_READ_DIR_FILELIST 22

#define F_OPEN_ONLY 		30
#define F_CREATE_ONLY 		31
#define F_WRITE_ONLY 		32
#define F_CLOSE_ONLY 		33

#define F_READ_FILES_CHAIN  40
#define F_EDIT_CHAIN  		41

#define F_SAVE_CURCFG_BIN		45
#define F_SAVE_AS_CURCFG_BIN	46
#define F_SAVE_SETUP_BIN		47
#define F_SAVE_AS_FULL_BIN	48

#define F_MODE_BINARY		0
#define F_MODE_XML			1
#define F_MODE_BINARY_FULL	2

typedef struct FILE_RW_typ
{

	USINT CMD;
	plcbit Done;
	plcbit Error;
	plcbit FileLocked;
	plcbit NewFileLoaded;
	USINT Mode;

	//plcstring varName[32];
	plcstring fileName[64];
	plcstring fileNewName[64];

	plcstring deviceName[32];
	plcstring targetDeviceName[32];

	plcstring MsgText[128];
	//FILE_SCHEDULE_typ FileSchedule;

	//CurCfg_typ curCfgTemp;
	//fiDIR_READ_DATA  FileInfo[1];

	TON_typ Tmr;

	UDINT pMem;
	UDINT Len;
	UDINT Offset;

	//XML_RW_HS_INT_typ _int;

}FILE_RW_typ;

typedef struct Calib_Param_typ
{
	UINT num;
	float val[8];

} Calib_Param_typ;

typedef struct CurCalib_typ
{
	UINT num;
	float TVL_Lo_Limit;
	float TVL_Hi_Limit;
	Calib_Param_typ Points[8];
	DINT GenSetup[8];
	float GenFloatValue[8];
	DINT  GenDintValue[8];
} CurCalib_typ;

/***********************************************/

/********			 Generic Motor 	    **********/

/***********************************************/
typedef struct GEN_MTR_msc_type
{

		AzzRamp_typ Ramp;

		AzzSlimPID_typ PID;
		azzslimpid_par_typ PIDParameters;

		/*
		LCRRamp_typ Ramp;

		LCRSlimPID_typ PID;
		lcrslimpid_par_typ PIDParameters;
		*/

		DINT Pos;
		INT _pos;
		float _vel;
		float _amp;
		float _volt;
		DINT deltaPos;

		//float kVel;
		//float kAcc;
		float kPos;

} GEN_MTR_msc_type;

typedef struct GEN_MTR_obj
{

	UDINT pState;
	plcstring Name[16];
	USINT Disable;
	USINT xCmd;
	float actPos;
	float actVel;
	float fParam[2];

	struct Hrdw
	{
		UINT *pPeriodDurationPWM;
		INT *pPulseWidthPWM;
		BOOL *pClearError;
		INT *pEncFbk;
		INT *pAnalogFbk;

	}Hrdw;

	struct Cfg{
		DINT units;
		float enc_dir;
		float mtr_dir;
		float rev_scale;
		//float loopPeriod;

	}Cfg;

	GEN_MTR_msc_type msc;

	/*
	struct msc
	{

		LCRRamp_typ Ramp;
		//LCRPT2o_typ Trajectory;
		//HCRFIFO_typ FIFODelay;
		//float FIFODelay[FIFO_DLY+1];

		LCRSlimPID_typ PID;
		lcrslimpid_par_typ PIDParameters;

		DINT Pos;
		INT _pos;
		float _vel;
		float _amp;
		float _volt;
		DINT deltaPos;

		//float kVel;
		//float kAcc;
		float kPos;

	} msc;
	*/

}GEN_MTR_obj;

///////////////////////////////////////////////////////////

typedef struct Cfg_DC2DIRMTR_obj{

	float MtrDir;
	BOOL *pQ1_output;
	BOOL *pQ2_output;
	BOOL *pQ3_output;
	BOOL *pQ4_output;

}Cfg_DC2DIRMTR_obj;

typedef	struct msc_DC2DIRMTR_obj
{
	UINT sw_step;

} msc_DC2DIRMTR_obj;

typedef struct DC2DIRMTR_obj
{
	UDINT pState;
	plcstring Name[16];
	USINT Disable;
	USINT xCmd;
	float fParam[2];
	Cfg_DC2DIRMTR_obj Cfg;
	msc_DC2DIRMTR_obj msc;

}DC2DIRMTR_obj;

typedef struct TML_OUTPUTS_Cfg_obj{

	float MtrDir;
	UINT TML_Vect_Indx;
	UINT TML_Indx;
	UINT Out1_Indx;
	UINT Out2_Indx;

}TML_OUTPUTS_Cfg_obj;

typedef	struct TML_OUTPUTS_msc_obj
{
	UINT sw_step;

} TML_OUTPUTS_msc_obj;

typedef struct TML_OUTPUTS_obj
{
	UDINT pState;
	plcstring Name[16];
	USINT Disable;
	USINT xCmd;
	float fParam[2];
	TML_OUTPUTS_Cfg_obj Cfg;
	TML_OUTPUTS_msc_obj msc;

}TML_OUTPUTS_obj;

//////////////////////////////////////////////////////////

/***********************************************/

/****        B&R 	Screen   						****/

/************************************************/

 //*===COLORS===*/
#define TRANSP						0xFF
#define GREEN						10
#define DARK_GREEN					2
#define BLUE						1
#define BABY_BLUE					11
#define TEAL						168
#define RED							0x33
#define YELLOW						46
#define BLACK						0
#define WHITE						15
#define GRAY						7
#define DARK_NAVY					219
#define DARK_GRAY					8
#define LIGHT_GRAY					227
#define CYAN						196
#define MAGENTA						21
#define BROWN						86
#define LIGHT_BLUE					52

typedef struct SCREEN_obj
{

	unsigned short SetPage;
	unsigned short ReadPage;
	unsigned short GotoScreen;
	unsigned short ReturnScreen;
	unsigned short Index;
	unsigned short NavMenu;
	unsigned short Update;
	plcbit btn_YES;
	plcbit btn_NO;
	plcbit btn[32];
	plcbit btnBar[32];
	plcbit btnMenu[10];
	plcbit btnSave;
	plcbit btnIndex;
	unsigned short vis[32];
	unsigned short visBar[32];
	unsigned short visSave;
	unsigned short colorBackground;
	unsigned short color[8];
	unsigned short colorBar[8];
	unsigned short colorSave;
	signed long Param[10];
	float fParam[10];
	unsigned short Language;
	unsigned short Units;
	unsigned short AngleUnits;
	float UnitsFactor;
	float UnitsOffset;
	unsigned long LifeSign;
	USINT AccessLevel;
	unsigned short menubtnColor[10];
  } SCREEN_obj;

/*
  typedef struct Screen_obj
{	unsigned short SetPage;
	unsigned short ReadPage;
	unsigned short GotoScreen;
	unsigned short ReturnScreen;
	unsigned short Index;
	unsigned short NavMenu;
	unsigned short Update;
	plcbit btn_YES;
	plcbit btn_NO;
	plcbit btnDefault;
	plcbit btn[32];
	plcbit btnGo2PrevScrn;
	plcbit RecipeModified;
	plcbit btnMoment[9];
	plcbit btnBar[32];
	plcbit btnMenu[20];
	plcbit btnSave;
	plcbit btnIndex;
	unsigned short vis[32];
	unsigned short visBar[32];
	unsigned short visSave;
	unsigned short colorBackground;
	unsigned short color[8];
	unsigned short colorBar[8];
	unsigned short colorSave;
	signed long Param[32];
	float fParam[20];
	plcstring stringParam[81];
	struct Pad_typ fPad[13];
	unsigned short fPadIndx;
	unsigned short ParamIndx;
	unsigned short fPad_vis;
	plcbit fPadUpdate;
	unsigned short Language;
	unsigned short LifeSign;
	unsigned short AccessLevel;
	unsigned short menubtnColor[10];
	unsigned char encIndex;
	unsigned char servoIndex;
}
*/
///////////////////////////////////////////////////////////

/***********************************************/

/****        Technosoft Servos					****/

/************************************************/

// Commands definition
#define TML_IDLE 0
#define TML_RESTART 1
// 2 - 13 reserved for TML_RESTART
#define TML_WAIT_FOR_DOWNLOAD 15
// 14 reserved for TML_RESTART
#define TML_HOLD_MODE 17
// 15 - 19 reserved for TML_HOLD_MODE
#define TML_POS_MODE 20
// 21 - 29 reserved for TML_POS_MODE
#define TML_VEL_MODE 30
// 31 - 39 reserved for TML_VEL_MODE
#define TML_TORQ_MODE 40
// 41 - 49 reserved for TML_TORQ_MODE
#define TML_VOLT_MODE 50
// 51 - 59 reserved for TML_VOLT_MODE
#define TML_PT_MODE 60
// 61 - 79 reserved for TML_PT_MODE
#define TML_CUST_MODE 80
// 81 - 89 reserved for TML_PT_MODE
#define TML_OSC_CUST_CMD 90
// 90 - 99 reserved for TML_PT_MODE
#define TML_DOWNL			100

/// New Osc

#define TML_SET_P_Max 		110
#define TML_SET_P_Min 		111
#define TML_SET_P_Time		112
#define TML_SET_P_DwellIn 	113
#define TML_SET_P_DwellOut 	114
#define TML_SET_P_Steer		115
#define TML_SET_P_Jog		117
#define TML_SET_P_Amplit 	118
#define TML_SET_Cmd_Word 	119

#define TML_SET_Cmd_Param 	120
#define TML_SET_Home 		121
#define TML_SET_Home2 		122

// New MIG Oscillator
#define TML_Cmd_SAP 		130
#define TML_Cmd_CPA			131
#define TML_Cmd_MODE_PP		132
#define TML_Cmd_TUM1 		133
#define TML_Cmd_CACC		134
#define TML_Cmd_CSPD		135
#define TML_Cmd_CPOS		136
#define TML_Cmd_UPD			137

///////////////////////////////
#define TML_KPP				140
#define TML_KIP				141
#define TML_KIP_Zero		145
#define TML_KPP_Zero		146
#define TML_SATP			150
#define TML_SATP_Zero		151

#define TML_UpdateFilter	160
#define TML_ClearFilter		161
#define TML_FullFilter		162
#define TML_SetGain			170

#define TML_SetGain_Zero	173

#define TML_MOVE_REL_CMD 175
// 175 - 190 reserved for TML_MOVE_REL_CMD

#define TML_RESET_ONLY_CMD 185
#define TML_FAULTR		   186

#define TML_ARC_CUST_CMD 190

#define TML_SET_OUT0_CMD 200
#define TML_RST_OUT0_CMD 201
#define TML_SET_OUT1_CMD 202
#define TML_RST_OUT1_CMD 203
#define TML_SET_OUT2_CMD 204
#define TML_RST_OUT2_CMD 205
#define TML_SET_OUT3_CMD 206
#define TML_RST_OUT3_CMD 207
#define TML_SET_OUT4_CMD 208
#define TML_RST_OUT4_CMD 209

#define TML_AXIS_ON_CMD  210
#define TML_AXIS_OFF_CMD 211

#define TML_UPD			212
#define TML_EINT		213

#define TML_MOVE_ABS_CMD 220

#define TML_READ_MCR 229

#define TML_UPD_CACC 230
#define TML_UPD_CSPD 231

// New MIG Oscillator Profile
#define TML_Cmd_OSC_Proc 235

#define TML_MOVE_ABS_PARM 245

////////

#define TML_DOWNL_DONE	222
#define TML_ERROR			255

// Status Mask
#define ERR_CANbus_MSK 			0x0001
#define ERR_ShortCircuit_MSK 	0x0002
#define ERR_InvalidSetup_MSK 	0x0004
#define ERR_Cntrl_MSK 			0x0008
#define ERR_RS232_MSK 			0x0010

//#define SREG_Fault_MSK 				0x80000000
#define SREG_Fault_MSK 				0x80000000

#define SREG_MotionCompleted_MSK 	0x00000400

//  Enumeration for new style OSC Parameters
#define V_Param_Cmd_Param	0
#define V_Param_Time 		1
#define V_Param_DwellIn 	2
#define V_Param_DwellOut 	3

#define V_fParam_Amplit 	0
#define V_fParam_Max 		1
#define V_fParam_Min 		2
#define V_fParam_Jog		3
#define V_fParam_Steer 		4
#define V_fParam_HomePos 	5

//  Enumeration for new MIG OSC Parameters

#define V_fParam_Cmd_SAP		0
#define V_fParam_Cmd_CPOS 		1
#define V_fParam_Cmd_CACC 		2
#define V_fParam_Cmd_CSPD 		3

//  Enumeration for new MIG OSC Profile

#define V_fParam_MIG_OSC_Amplit		0
#define V_fParam_MIG_OSC_Speed 		1
#define V_fParam_MIG_OSC_Acc		2
#define V_fParam_MIG_OSC_DwellIn 	3
#define V_fParam_MIG_OSC_DwellOut	4

//  Enumeration for Rel Move Parameters

#define V_fParam_Rel_CACC		0
#define V_fParam_Rel_CSPD 		1
#define V_fParam_Rel_CPOS 		2

/////////////////////////////////////////
/******  TML STatus enumeration    *****/

typedef enum TML_STAT_Enum
{
	TML_STAT_DRIVE_ERR = 	-4,
	TML_STAT_VER_ERR   =	-3,
	TML_STAT_INIT  	   =	-2,
	TML_HEARTBEAT_ERR  = 	-1,
	TML_STAT_DEAD  	   =	0,
	TML_STAT_READY 	   =	1,
	TML_STAT_IDLE 	   =	2,
	TML_STAT_HOLD_INIT 	   =	3,
	TML_STAT_HOLD_OK 	   =	4,
	TML_STAT_POS_MODE_INIT  =	5,
	TML_STAT_POS_MODE_OK    =	6,
	TML_STAT_VEL_MODE_INIT  =	7,
	TML_STAT_VEL_MODE_OK 	=	8,
	TML_STAT_TORQ_MODE_INIT =	9,
	TML_STAT_TORQ_MODE_OK 	=	10,
	TML_STAT_VOLT_MODE_INIT =	11,
	TML_STAT_VOLT_MODE_OK 	=	12,
	TML_STAT_PT_MODE_INIT 	=	13,
	TML_STAT_PT_MODE_OK 	=	14,
	TML_STAT_CUSTOM_INIT 	   =	15,
	TML_STAT_CUSTOM_OK 	   =	16,
	TML_STAT_DRIVE_SELF_CNTRL 	   =	17,

}TML_STAT_Enum;

typedef struct TML_typ
{
	StateVectorProxy_typ* pState;
	plcstring Name[16];
	USINT Disable;
	unsigned long  ProgramVersion;
	unsigned long  FirmwareVersion;

	float PosFBK;
	USINT xCMD;
	TML_STAT_Enum Status;
	unsigned long StatusReg;
	unsigned short ErrorReg;
	unsigned short MCRReg;
	plcbit Error;
	plcbit EnableInp;
	unsigned short AnInp[2];
	plcbit DigInp[4];
	plcbit DigOut_stat[4];
	plcbit EStop;

	plcbit HoldErrorReg;

	// DigInp[2] = LSP
	// DigInp[3] = LSN
	// AnInp[0] = REF
	// AnInp[1] = FDBK
	struct _cfg{
		DINT units;
		float rev_motor;
		float rev_scale;
		float actPos2_scale;
		UINT  absFbk;
		DINT absLastPos;
		DINT *pAbsLastPos;
		float loopPeriod;
		float maxVel;
		float maxAcc;
		float signFilter;
		//DINT  satp;
		DINT  satpMax;
		DINT  kip;
		DINT  kipMax;
		DINT  kpp;
		DINT  kppMax;
		DINT  SATSMax;
		plcstring programName[32];
		float HeartBeat;
		float PVTPeriod;
		UINT MtrType;
		//float sftLimitPos;
		//float sftLimitNeg;
		UINT NotAutoDownload;
		UDINT Appl_ID_adr;
		unsigned short AnalLimitPos;
		unsigned short AnalLimitNeg;

	}_cfg;

	struct _int{
		DINT _pos;
		DINT _deltaPos;
		UINT _posCnt;
		float _floatPos;
		float _vel;
		float _amp;
		float _volt;
		float kVel;
		float kAcc;
		float kPos;
		float kVolt;
		UINT PVTPeriod;
		SINT Init;
		float startPos;
		UINT restartCnt;
		UINT cnt;
		//UINT msgProcess;
		UINT KickCntr;
		DINT const_PT;
		TON_typ dly_Tmr;

	}_int;

} TML_typ;

typedef struct TML_CHAN_HRDW_typ
{
	USINT AxisNum;

	USINT TXCountReadBack;
	//
	USINT RXDataSize0;
	USINT RXCount;
	USINT buff[4];
	UDINT RXIdent0;
	UINT  RXData0Word0[4];
	//
	USINT TXCount;
	USINT TXDataSize;
	UDINT TXIdent;
	UINT  TXDataWord0[4];

	USINT _oldRxCount;
	USINT _indx;

	TON_typ DlyTmr;

}TML_CHAN_HRDW_typ;

typedef struct TML_Axis_typ
{	unsigned short AxisID;
	unsigned long  Version;
	unsigned long  ProgramVersion;
	unsigned long  FirmwareVersion;
	USINT  Flag;
	UINT  AxisState;
	unsigned short DriveStatusRegisterL;
	unsigned short DriveStatusRegisterH;
	unsigned short DriveErrorRegister;
	unsigned short PVTstatus;
	unsigned short DataLow;
	unsigned short DataHigh;
	unsigned short VarAddress;
	unsigned short SATS;
	signed long	   curPos;
	signed long	   _curPos;
	signed long	   _lastPos;
	unsigned short pointer;
	short deltaAPOS;
	//unsigned long  CmdWord;
	unsigned short PointCounter;
	TON_typ HeartBeat;
	TON_typ InitTmr;

} TML_Axis_typ;

typedef struct TML_MGR_typ
{
	UDINT pSendData[2]; // two channels
	UDINT pRecData[2]; // two channels
	TML_CHAN_HRDW_typ hrdw[2];
	UDINT Firmware[2];
	USINT BlockTrans[2];
	TML_Axis_typ *pAxis[2];
	TML_typ *pTML[2];
	UDINT pLog;

}TML_MGR_typ;

///////////////////////////////////////////////////////////

typedef struct SerialPortDriver{
	 FRM_xopen_typ	 Open;
	 XOPENCONFIG	 OpenConfig;
	 FRM_gbuf_typ	 GetBuffer;
	 FRM_rbuf_typ	 Release;
	 FRM_robuf_typ	 ReleaseOutput;
	 FRM_write_typ	 Write;
	 FRM_read_typ	 Read;
	 FRM_mode_typ	 Mode;
	 FRM_close_typ	 Close;

	 UINT			 StatusOpen;
	 UINT			 StatusWrite;
	 UINT			 StatusRead;
	 UINT			 StatusGetBuffer;
	 UINT			 StatusReleaseOutputBuffer;
	 UINT			 StatusMode;
	 UINT			 StatusClose;

	 UDINT			 Ident;
	 UDINT* 		 pSendBuffer;
	 UDINT* 		 pReadBuffer;
	 UINT			 SendLength;
	 UINT			 ReadLength;
	 UINT			 l;

	 UINT			 txRequest;
	 UINT			 txBufRequest;
	 UINT			 txDataLen;
	 UINT			 rxReady;
	 UINT			 txMessageCounter;
	 UINT			 rxMessageCounter;
	 UINT			 txError;
	 UINT			 rxError;
	 UINT			 initError;

	 STRING 		 sDevice[32];
	 STRING 		 sMode[64];
	 STRING 		 sModeNew[64];
	 USINT			 _parity;

	 plcstring		 txData[256];
	 plcstring		 rxData[256];
	 STRING 		 sInput[64];

 }SerialPortDriver_typ;
 /***************************************/

/////////////////////////////////////////////////////
///   New Path Generator created March 2019 by CK
/////////////////////////////////////////////////////

/////////////////////////////////////////////////////

typedef struct HCRMoveParamAzz_type
{
	float t_Jolt;
	float vC_pos;
	float vC_neg;
	float aAcc_pos;
	float aDec_pos;
	float aAcc_neg;
	float aDec_neg;
} HCRMoveParamAzz_type;

typedef struct segment_type{

	float s;
	float a;
	float v;

}segment_type;

typedef struct HCRSPFazz_Internal_type
{
	plcstring statusTxt[81];
	UINT step;

	float S0;
	float S1;
	float S2;
	float S3;

	float _s_set;
	float _v_set;
	float _a_set;
	UINT _uSec;
	UINT uSec;
	UINT indx;

	plcbit _enable;
	plcbit _Stop;
	plcbit _Set_home;
	plcbit _Init;
	plcbit _Brake;

	float vC_pos;
	float vC_neg;
	float aAcc_pos;
	float aDec_pos;
	float aAcc_neg;
	float aDec_neg;

	float TaskPeriod;

	segment_type segm[4];

}HCRSPFazz_Internal_type;

typedef struct HCRMoveParaAzz_type
{
	float t_Jolt;
	float vC_pos;
	float vC_neg;
	float aAcc_pos;
	float aDec_pos;
	float aAcc_neg;
	float aDec_neg;
} HCRMoveParaAzz_type;

typedef struct HCRSPFazz_type
{
	/* VAR_INPUT (analog) */
	//struct HCRMovePara_typ* pMove_Para;
	struct  HCRMoveParamAzz_type* pMove_Para;
	float s_home;
	float s_end;
	/* VAR_OUTPUT (analog) */
	float s_set;
	float v_set;
	float a_set;
	float elapseTime;
	signed char MoveDir;
	signed char ApproachDir;
	unsigned short status;
	/* VAR (analog) */
	struct HCRSPFazz_Internal_type Intr;
	/* VAR_INPUT (digital) */
	plcbit enable;
	plcbit Stop;
	plcbit Set_home;
	plcbit Init;
	plcbit Brake;
	/* VAR_OUTPUT (digital) */
	plcbit Reached;
} HCRSPFazz_type;

#endif
```

### xstring.c
```c
#ifndef _XTRINGLIB_C
#define _XTRINGLIB_C

#include <stdarg.h>
//#include <stdlib.h>
//#include <string.h>
#include <ctype.h>
#include <math.h>

int xputs(int c, char **where);

int xpadit(int n, int c, int (*put)(), char **where);

int xprint(int (*put)(), char **where, char *fmt, va_list varg);
int pprint(int (*put)(), char **where, char *fmt, va_list varg);

int  xuxtoi(char *str);
long xuxtol(char *str);
int xatoi(char *str);
long xatol(char *str);

char *xultoa(unsigned long val, int base, int convup);
char *xfdtoa(double fval, int prec);
char *xftoa(float fval, int prec);

int xsprintf(char *where, char *fmt, ...);
int psprintf(char *where, char *fmt, ...);

/**************************************************************************/

#define CHRSTR          0       /* type is char or string*/
#define DOUX            1       /* type is d, o, u, x, X*/
#define CONVE           2       /* type is e, E*/
#define CONVF           3       /* type is f*/
#define CONVG           4       /* type is g,G*/
#define SIGN_OK         0       /* Signed*/
#define UNSIGN_OK       4       /* Unsigned*/

/***********/
int xputs(int c, char **where)
{
  return(*(*where)++ = c);
}
/***********/

/* Put out n characters.  No characters will be output if n <= 0.*/
int xpadit(int n, int c, int (*put)(), char **where)
{
  while(n-- > 0)
  {
    if ((*put)(c, where) != c)
    {
      return 1;
    }
  }
  return 0;
}
/***********/

char *xsltoa(long val, int base, int convup)
{
  static char buf[32];
  char sign = '+';
  char *p;
  char *str;

  if (val < 0)
  {
    val = -val;
    sign = '-';
  }

  str = convup?"0123456789ABCDEF":"0123456789abcdef";

  p = buf+31;
  *p = 0;

  do
  {
    *--p = str[val % base];
  } while(val /= base);

  *--p = sign;
  return p;
}

/***********/

char *xultoa(unsigned long val, int base, int convup)
{
  static char buf[32];
  char *p;
  char *str;
  char leadZero;

  str = convup?"0123456789ABCDEF":"0123456789abcdef";

  p = buf+31;
  *p = 0;

  leadZero = (val < base)? 1:0;

  do
  {
    *--p = str[val % base];
  } while(val /= base);

  if(leadZero)
  	 *--p = str[0];

  return p;
}
/**********************/

char *xfdtoa(double fval, int prec)
{

double rem, integ , _fval;
unsigned long	val , _val ;
static char buf[32];
char *p;
char *str;
double _pow;

	str = "0123456789ABCDEF";

	p = buf+31;
	*p = 0;

	if(prec>0){

		rem = modf (fabs(fval),&integ);

		_pow = powf(10.0 , (double)prec);

		val = (unsigned long)(rem * _pow + 0.5);
		_val = val;

		do
		{
			*--p = str[val % 10];
			val /= 10;
		} while(--prec>0);

		*--p = '.';

		val = (unsigned long)integ + _val/_pow;

	}
	else
		val = ((unsigned long)(fabs(fval)*10 + 5))/10 ;

	do
	{
	*--p = str[val % 10];
	}  while(val /= 10);

	if(fval<0)
		*--p ='-';
	else if(fval>0)
		*--p ='+';

  return p;
}

char *xftoa(float fval, int prec)
{ float rem, integ;
  unsigned long	val;
  static char buf[32];
  char *p;
  char *str;

  str = "0123456789ABCDEF";
  p = buf+31;
  *p = 0;

	rem = modff (fabsf(fval),&integ);

	if(prec>0){
		val = (unsigned long)(rem * ( (float)powf(10.0 , (double)prec))+0.5);

		do
		{
			*--p = str[val % 10];
		} while(val /= 10);

		*--p = '.';

	}

	val = (unsigned long)integ;

	do
	{
		*--p = str[val % 10];
	}  while(val /= 10);

	if(fval<0)
		*--p ='-';

  return p;
}

/***********/
int xprint(int (*put)(), char **where, char *fmt, va_list varg)
{
  int  c;
  int  zeros, left, sign, blank, alternate, longarg;
  int  width, precision, len, pad, prpad, prtsign, numalt, prttype;
  int  retv, getwidth, getprec, convup, padzero;
  long val;
  char *p;
  char buf[3];
  double fval;

  /*Valid printf characters (in specific order).*/
  static char validc[] = "douxXcsfeEgG";

  retv   = 0;
  buf[1] = 0;

  for (; (c=*fmt); ++fmt)
  {
      /* If the character's not a % or if it is a %% then just put out the character and continue.*/
      if ((c != '%') || ((c = *++fmt) == '%'))
      {
        ++retv;
        if ((*put)(c, where) != c)
        {
          return -1;
        }
        continue;
      }

      zeros = left = sign = blank = alternate = 0;

      do
      {
        if (c == '-')
          left = 1;
        else if (c == '+')
          sign = 1;
        else if (c == ' ')
          blank = 1;
        else if (c == '#')
          alternate = 1;
        else if (c == '0')
          zeros = 1;
        else
          break;
      }
      while (c = *++fmt);

      width = -1;
      if (getwidth = (c == '*'))
      {
        c = *++fmt;
      }
      else if (isdigit(c))
      {
        width = xatoi(fmt);
        while (c = *++fmt, isdigit(c))
        {
        }
      }

      getprec   = 0;
      precision = -1;
      if (c == '.')
      {
        c = *++fmt;
        if (getprec = (c == '*'))
        {
          c = *++fmt;
        }
        else
        {
          precision = xatoi(fmt);
          while(isdigit(c))
          {
            c = *++fmt;
          }
        }
      }

      if (longarg = (c == 'l'))
      {
        c = *++fmt;
      }

      padzero = 1;
      convup = numalt = prtsign = 0;

      if (p = strchr(validc, c))
      {
        if (getwidth)
        {
          width = va_arg(varg, int);
        }

        if (getprec)
        {
          precision = va_arg(varg, int);
        }

		if(c== 'f'){
			fval =(float) va_arg(varg, double);
		}
        else if (p == (validc + SIGN_OK) )
        {
          val = (longarg?va_arg(varg, long):(long)va_arg(varg, int));
        }
        else if (p <= (validc + UNSIGN_OK))
        {
          val = (longarg?va_arg(varg, unsigned long):(long)va_arg(varg, unsigned int));
        }
      }

      switch(c)
      {
        case 'f':
            p = xfdtoa(fval, precision);
			prtsign = *p++;
            if (!sign && (prtsign == '+'))
            {
              prtsign = (blank?' ':0);
            }
            prttype = DOUX;
            break;
        case 'd':
            p = xsltoa(val, 10, 0);
            prtsign = *p++;
            if (!sign && (prtsign == '+'))
            {
              prtsign = (blank?' ':0);
            }
            prttype = DOUX;
            break;

        case 'o':
            p = xultoa(val, 8, 0);
            numalt = 1;
            prttype = DOUX;
            break;
        case 'u':
            p = xultoa(val, 10, 0);
            prttype = DOUX;
            break;
        case 'X':
            convup = 1;
            /*fall thru*/
        case 'x':
            p         = xultoa(val, 16, convup);
            numalt    = 2;
            prttype   = DOUX;
            break;
        case 's':
            p         = va_arg(varg, char*);
            prttype   = CHRSTR;
            break;
        case 'c':
            c         = va_arg(varg, int);
            c         &= 0x00ff;
            /*fall thru*/
        default:
            buf[0]    = c;
            p         = buf;
            precision = 1;
            prttype   = CHRSTR;
      }

	 /*Handle the final printing of conversions for f*/
      if (prttype == CONVF)
      {
	  	 p = xfdtoa(fval, precision);
            prtsign = *p++;
            if (!sign && (prtsign == '+'))
            {
              prtsign = (blank?' ':0);
            }
            prttype = DOUX;
      }
    /*Handle the final printing of conversions for d,o,u,x,X*/
      if (prttype == DOUX)
      {
        if (val == 0)
        {
          alternate = 0;
          if (precision == 0)
          {
            *p = 0;
          }
        }

        len = strlen(p);

        if ((prpad = precision - len) > 0)
        {
          if (alternate && (numalt == 1))
          {
            --prpad;
          }
        }
        else
        {
          prpad = 0;
        }

        pad = width - len - prpad;

        if (alternate)
        {
          pad -= numalt;
        }

        if (prtsign)
        {
          --pad;
        }

        if (pad < 0)
        {
           pad = 0;
        }

        retv += len + pad + prpad;

        if (zeros)
        {
          if (!left && xpadit(pad, '0', put, where))
          {
            return -1;
          }
        }
        else
        {
          if (!left && xpadit(pad, ' ', put, where))
          {
            return -1;
          }
        }

        if (prtsign)
        {
          if ((*put)( prtsign, where ) != prtsign)
          {
            return -1;
          }
          ++retv;
        }

        if (alternate && numalt)
        {
          if ((*put)('0', where) != '0')
          {
            return -1;
          }
          retv += numalt;
          if ((numalt == 2) && ((*put)(c, where) != c))
          {
            return -1;
          }
        }

        if (xpadit(prpad, '0', put, where))
        {
          return -1;
        }
        while (c = *p++)
        {
          if ((*put)(c, where) != c)
          {
            return -1;
          }
        }
        if (left && xpadit(pad, ' ', put, where))
        {
          return -1;
        }
      }
      else if (prttype == CHRSTR)
      {
      	if(p)
        	len = strlen(p);
		else
			len = 0;

        if ((precision != -1) && (precision < len))
        {
          len = precision;
        }

        if ((pad = width - len) < 0)
        {
          pad = 0;
        }

        retv += width + pad;

        if (!left && xpadit(pad, ' ', put, where))
        {
          return -1;
        }

        while (width-- && (c = *p++))
        {
          if ((*put)(c, where) != c)
          {
            return -1;
          }
        }
        if (left && xpadit(pad, ' ', put, where))
        {
          return -1;
        }
      }
  }

  return retv;
}
/****************************/
int pprint(int (*put)(), char **where, char *fmt, va_list varg)
{
  int  c;
  int  zeros, left, sign, blank, alternate, longarg;
  int  width, precision, len, pad, prpad, prtsign, numalt, prttype;
  int  retv, getwidth, getprec, convup, padzero;
  long val;
  unsigned long *pval;
  char *p;
  char buf[3];
  double fval;
  float *pfval;
  unsigned long pointer;

  /*Valid printf characters (in specific order).*/
  static char validc[] = "douxXcsfeEgG";

  retv   = 0;
  buf[1] = 0;

  for (; (c=*fmt); ++fmt)
  {
      /* If the character's not a % or if it is a %% then just put out the character and continue.*/
      if ((c != '%') || ((c = *++fmt) == '%'))
      {
        ++retv;
        if ((*put)(c, where) != c)
        {
          return -1;
        }
        continue;
      }

      zeros = left = sign = blank = alternate = 0;

      do
      {
        if (c == '-')
          left = 1;
        else if (c == '+')
          sign = 1;
        else if (c == ' ')
          blank = 1;
        else if (c == '#')
          alternate = 1;
        else if (c == '0')
          zeros = 1;
        else
          break;
      }
      while (c = *++fmt);

      width = -1;
      if (getwidth = (c == '*'))
      {
        c = *++fmt;
      }
      else if (isdigit(c))
      {
        width = xatoi(fmt);
        while (c = *++fmt, isdigit(c))
        {
        }
      }

      getprec   = 0;
      precision = -1;
      if (c == '.')
      {
        c = *++fmt;
        if (getprec = (c == '*'))
        {
          c = *++fmt;
        }
        else
        {
          precision = xatoi(fmt);
          while(isdigit(c))
          {
            c = *++fmt;
          }
        }
      }

      if (longarg = (c == 'l'))
      {
        c = *++fmt;
      }

      padzero = 1;
      convup = numalt = prtsign = 0;

      if (p = strchr(validc, c))
      {
        if (getwidth)
        {
          width = va_arg(varg, int);
        }

        if (getprec)
        {
          precision = va_arg(varg, int);
        }

		if(c!= 's'){

			pointer = va_arg(varg, unsigned long);

			if(!pointer)
				return;
		}

      }

      switch(c)
      {
        case 'f':

			pfval = pointer;

			p = xfdtoa(*pfval, precision);
			prtsign = *p++;
            if (!sign && (prtsign == '+'))
            {
              prtsign = (blank?' ':0);
            }
            prttype = DOUX;
            break;
        case 'd':

			pval = pointer;

            p = xsltoa(*pval, 10, 0);
            prtsign = *p++;
            if (!sign && (prtsign == '+'))
            {
              prtsign = (blank?' ':0);
            }
            prttype = DOUX;
            break;

        case 'o':

			pval = pointer;

            p = xultoa(*pval, 8, 0);
            numalt = 1;
            prttype = DOUX;
            break;
        case 'u':

			pval = pointer;

            p = xultoa(*pval, 10, 0);
            prttype = DOUX;
            break;
        case 'X':
            convup = 1;
            /*fall thru*/
        case 'x':

			pval = pointer;
            p         = xultoa(*pval, 16, convup);
            numalt    = 2;
            prttype   = DOUX;
            break;
        case 's':
            p         = va_arg(varg, char*);
            prttype   = CHRSTR;
            break;
        case 'c':
            c         = va_arg(varg, int);
            c         &= 0x00ff;
            /*fall thru*/
        default:
            buf[0]    = c;
            p         = buf;
            precision = 1;
            prttype   = CHRSTR;
      }

	 /*Handle the final printing of conversions for f*/
      if (prttype == CONVF)
      {
	  	 p = xfdtoa(fval, precision);
            prtsign = *p++;
            if (!sign && (prtsign == '+'))
            {
              prtsign = (blank?' ':0);
            }
            prttype = DOUX;
      }
    /*Handle the final printing of conversions for d,o,u,x,X*/
      if (prttype == DOUX)
      {
        if (val == 0)
        {
          alternate = 0;
          if (precision == 0)
          {
            *p = 0;
          }
        }

        len = strlen(p);

        if ((prpad = precision - len) > 0)
        {
          if (alternate && (numalt == 1))
          {
            --prpad;
          }
        }
        else
        {
          prpad = 0;
        }

        pad = width - len - prpad;

        if (alternate)
        {
          pad -= numalt;
        }

        if (prtsign)
        {
          --pad;
        }

        if (pad < 0)
        {
           pad = 0;
        }

        retv += len + pad + prpad;

        if (zeros)
        {
          if (!left && xpadit(pad, '0', put, where))
          {
            return -1;
          }
        }
        else
        {
          if (!left && xpadit(pad, ' ', put, where))
          {
            return -1;
          }
        }

        if (prtsign)
        {
          if ((*put)( prtsign, where ) != prtsign)
          {
            return -1;
          }
          ++retv;
        }

        if (alternate && numalt)
        {
          if ((*put)('0', where) != '0')
          {
            return -1;
          }
          retv += numalt;
          if ((numalt == 2) && ((*put)(c, where) != c))
          {
            return -1;
          }
        }

        if (xpadit(prpad, '0', put, where))
        {
          return -1;
        }
        while (c = *p++)
        {
          if ((*put)(c, where) != c)
          {
            return -1;
          }
        }
        if (left && xpadit(pad, ' ', put, where))
        {
          return -1;
        }
      }
      else if (prttype == CHRSTR)
      {
		if(p)
			len = strlen(p);
		else
			len = 0;

        if ((precision != -1) && (precision < len))
        {
          len = precision;
        }

        if ((pad = width - len) < 0)
        {
          pad = 0;
        }

        retv += width + pad;

        if (!left && xpadit(pad, ' ', put, where))
        {
          return -1;
        }

        while (width-- && (c = *p++))
        {
          if ((*put)(c, where) != c)
          {
            return -1;
          }
        }
        if (left && xpadit(pad, ' ', put, where))
        {
          return -1;
        }
      }
  }

  return retv;
}

/***********/

int  xuxtoi(char *str)
{
  int  num;
  char c;

  c = *str;
  while ((c==' ') || (c=='\t'))
  {
    ++str;
  }

  for(num=0; isxdigit(c); c=*++str)
  {
    if (c<='9')
      c -= '0';
    else if (c<='F')
      c = (c-'A')+10;
    else
      c = (c-'a')+10;

    num = (num*16) + (int)c;
  }

  return(num);
}

/***********/

long xuxtol(char *str)
{
  long num;
  char c;

  c = *str;
  while ((c==' ') || (c=='\t'))
  {
    ++str;
  }

  for(num=0; isxdigit(c); c=*++str)
  {
    if (c<='9')
      c -= '0';
    else if (c<='F')
      c = (c-'A')+10;
    else
      c = (c-'a')+10;

    num = (num*16) + (long)c;
  }

  return(num);
}

/***********/

int xatoi(char *str)
{
  int  num;
  int  neg;
  char c;

  c = *str;

  while ((c == ' ') || (c == '\t'))
  {
    ++str;
  }

  if (*str == '-')
  {
    neg = 1;
    ++str;
  }
  else
  {
    neg = 0;
  }

  for(num=0; isdigit(c); c = *++str)
  {
    num = (num*10) + (c -= '0');
  }

  if (neg)
  {
    return(-num);
  }
  else
  {
    return(num);
  }
}

/***********/

long xatol(char *str)
{
  long num;
  int  neg;
  char c;

  c = *str;

  while ((c == ' ') || (c == '\t'))
  {
    ++str;
  }

  if (*str == '-')
  {
    neg = 1;
    ++str;
  }
  else
  {
    neg = 0;
  }

  for(num=0; isdigit(c); c = *++str)
  {
    num = (num*10) + (long)(c -= '0');
  }

  if (neg)
  {
    return(-num);
  }
  else
  {
    return(num);
  }
}
/************************************/
int xsprintf(char *where, char *fmt, ...)
{
  int     retv;
  va_list varg;

  va_start(varg, fmt);
  retv = xprint(xputs, &where, fmt, varg);
  *where = 0;
  va_end(varg);

  return retv;
}
/************************************/
int psprintf(char *where, char *fmt, ...)
{
  int     retv;
  va_list varg;

  va_start(varg, fmt);
  retv = pprint(xputs, &where, fmt, varg);
  *where = 0;
  va_end(varg);

  return retv;
}

#endif
```

### LoggerLib.c
```c
/********************************************************************
 * COPYRIGHT -- PAI
 ********************************************************************
 * Library: Logger
 * File: LoggerLib.c
 * Author: Christopher
 * Created: December 26, 2008
 *******************************************************************/
#ifndef _LOGGERLIB_C
	#define _LOGGERLIB_C

#include <bur/plctypes.h>

#include <..\Lib\LoggerLib.h>

	USINT buf1[MAXLOGS * ((MAXLOGINPUT+1) + sizeof(plcdt)+ sizeof(plctime))];
	USINT buf2[MAXLOGS * ((MAXLOGINPUT+1) + sizeof(plcdt)+ sizeof(plctime))];

	void SetTimeStamp(plctime t , plcdt dt, char * p , char * txt);

	//#include <..\globalvar.h>

	DINT LoggerInit(LOGMGR_obj *log ,UDINT *Id, char *dbName , UINT maxLogs){

		log->_int.MaxLogs = maxLogs;

		if(dbName == 0) if(Id == 0) return -200;

		// New 8 Nov 19
		if(*Id > maxLogs)
			*Id = 0;
		//////////////

		strcpy ( log->_int.dbName , dbName);
		if(Id == 0) return -100;
		log->_int.pLogID  = (UDINT*) Id;

		log->_int.recLen = MAXLOGINPUT + sizeof(plcdt)+ sizeof(plctime);

		/* Initialize info structure */
		log->_int.DOInfo.enable   		= 1;
		log->_int.DOInfo.pName    		= (UDINT) log->_int.dbName;
		/***/

		/* Call  FUB  */
		/***/
		DatObjInfo(&log->_int.DOInfo);
		log->_int.Status 	= log->_int.DOInfo.status;

		if (log->_int.Status == doERR_MODULNOTFOUND)  {
			log->_int.DataObjReady	= 0;
			log->Ready				= 0;
			log->_int.WriteData		= 0;
			log->_int.ReadData		= 0;
			log->_int.Create 		= 1;
			return -1;
		}
		else if( log->_int.MaxLogs * (sizeof( log->Logtxt_inp) + sizeof(plcdt) + sizeof(plctime)) != log->_int.DOInfo.len){
			log->_int.DataObjReady	= 0;
			log->Ready				= 0;
			log->_int.WriteData		= 0;
			log->_int.ReadData		= 0;
			log->_int.Create 		= 0;
			return -2;

		}
		else {
			log->_int.DataObjReady	= 1;
			log->Ready				= 1;
			log->_int.WriteData		= 0;
			log->_int.ReadData		= 1;
			log->_int.Create 		= 0;
			log->_int.dwIdent 		= log->_int.DOInfo.ident;
			return 1;

		}
	}

	DINT LoggerSrv(LOGMGR_obj *log ){
	INT i , j , k , l;
	DTGetTime_typ DTGetTime_1;
	DTStructure _DTStruct;
	plcdt		_dt;
	plctime _t;
	char _buf[50];
	char *p;
	UDINT buf1Len , buf2Len , buf1Offset , buf2Offset;

		// New 8 Nov 19
		if(!log->_int.pLogID)
			return -1;

		if(*log->_int.pLogID > log->_int.MaxLogs)
			*log->_int.pLogID = 0;
		////////////////////

		if( log->Cmd.EraseAllLogs)  {
			log->Cmd.EraseAllLogs = 0;
			log->_int.Create = 1;
			log->Cmd.Refresh = 1;

		}

		if ( log->_int.Create )  {
			(*log->_int.pLogID) = 0;
		   	log->_int.DOCreate.enable	   = 1;
		   	log->_int.DOCreate.grp 	   = 0;
		   	log->_int.DOCreate.pName	   = (UDINT) log->_int.dbName;
		   	log->_int.DOCreate.len 	   =  log->_int.MaxLogs * (sizeof( log->Logtxt_inp) + sizeof(plcdt)+ sizeof(plctime));
		   	log->_int.DOCreate.MemType    = doUSRROM;
		   	log->_int.DOCreate.Option	   = 0;
		   	log->_int.DOCreate.pCpyData   = 0;

		   	/* Call FUB */
		   	DatObjCreate(&log->_int.DOCreate);
		   	log->_int.Status   = log->_int.DOCreate.status;
		   	log->_int.dwIdent			   = log->_int.DOCreate.ident;

		   	/* Verify status */
		   	if (log->_int.Status == 0) {
			   log->_int.DataObjReady 	= 1;
			   log->Ready				= 1;
		   	}
			else if(log->_int.Status == 65535) return 0; /** Function Busy - try again **/
		   	else if (log->_int.Status != 0xFFFF) {
		   	}
			log->_int.Create = 0;
		 }

		 if(!log->_int.DataObjReady) return -100;

		/** *******************************/
		if(log->Cmd.EnterLog ){
			log->Cmd.EnterLog = 0;

			if(log->Cmd.PauseLog) return 100;

			/* Get Date Time String */
			DTGetTime_1.enable = 1;
			DTGetTime(&DTGetTime_1);

			memset(log->_int.logBuf , 0 , sizeof(log->_int.logBuf));
			memcpy(log->_int.logBuf , &DTGetTime_1.DT1 , sizeof(plcdt));
			_t = clock_ms();
			memcpy(log->_int.logBuf + sizeof(plcdt) ,&_t , sizeof(plctime));

			if(strlen(log->Logtxt_inp) >= MAXLOGINPUT)
				log->Logtxt_inp[MAXLOGINPUT-1] = 0;

			strcpy(log->_int.logBuf + sizeof(plcdt)+ sizeof(plctime) , log->Logtxt_inp);

			/*
			if(strlen(log->Logtxt_inp)< MAXLOGINPUT)
				strcpy(log->_int.logBuf + sizeof(plcdt)+ sizeof(plctime) , log->Logtxt_inp);
			else
				strcpy(log->_int.logBuf , "log txt too long ");
			*/

			log->_int.DOWrite.enable	= 1;
		   	log->_int.DOWrite.ident		= log->_int.dwIdent;
		   	log->_int.DOWrite.Offset	= (*log->_int.pLogID)  * log->_int.recLen;
		   	log->_int.DOWrite.pSource	= (UDINT)log->_int.logBuf ;
		   	log->_int.DOWrite.len		= log->_int.recLen;

		   	/* Call FUB */
		    DatObjWrite(&log->_int.DOWrite);
		   	log->_int.Status   = log->_int.DOWrite.status;
			if(log->_int.Status == 20605){
				LoggerInit(log , log->_int.pLogID , log->_int.dbName , log->_int.MaxLogs);
				return 1;
			}
			else if(log->_int.Status == 65535) return 0; /** Function Busy - try again **/
				log->Cmd.EnterLog = 0;

			if(log->_int.Status == 0){
				(*log->_int.pLogID) ++;
				SetTimeStamp(_t ,DTGetTime_1.DT1,log->LastLog , log->Logtxt_inp);

			}
			if((*log->_int.pLogID)> (log->_int.MaxLogs-1)) (*log->_int.pLogID) = 0;
				log->_int.DOWrite.enable	= 0;

			if(!log->Cmd.PauseRefreshNewLog)log->Cmd.Refresh = 1;

		}

		if((log->Cmd.scrollBy > log->_int.MaxLogs) ||
			(log->Cmd.scrollBy == 0)) log->Cmd.scrollBy = 1;

		if(log->Cmd.ScrollUp){
			log->Cmd.ScrollUp = 0;
			log->curLog -= log->Cmd.scrollBy ;
			log->Cmd.Refresh = 1;
		}

		if(log->Cmd.ScrollDwn){
			log->Cmd.ScrollDwn = 0;
			log->curLog += log->Cmd.scrollBy ;
			log->Cmd.Refresh = 1;
		}

		if(log->Cmd.LastLogs){
			log->Cmd.LastLogs = 0;
			log->curLog = 0;
			log->Cmd.Refresh = 1;
		}

		if(log->Cmd.Refresh){

			if(log->Cmd.PauseRefresh){
				log->Cmd.Refresh = 0;
				return 101;
			}

			if(log->curLog > log->_int.MaxLogs) log->curLog = 0;

			if((*log->_int.pLogID) >= (log->curLog  + MAXLOGS)){
				buf1Len 	= MAXLOGS;
				buf1Offset 	= ((*log->_int.pLogID)  - log->curLog -  MAXLOGS) * log->_int.recLen ;
				buf2Len 	= 0;
				buf2Offset 	= 0;
			}

			else {
				if((*log->_int.pLogID)  >= log->curLog){
					buf1Len 	= (*log->_int.pLogID)  -  log->curLog;
					buf1Offset 	= 0;
					buf2Len 	= MAXLOGS - buf1Len;
					buf2Offset 	= (log->_int.MaxLogs - buf2Len ) * log->_int.recLen;
				}
				else{
					buf1Len 	= 0;
					buf1Offset 	= 0;
					buf2Len		= MAXLOGS;
					buf2Offset	=(log->_int.MaxLogs - (log->curLog - (*log->_int.pLogID)) - MAXLOGS) * log->_int.recLen;
				}
			}

			memset(&log->LogView , 0 , sizeof(log->LogView));
			k = 0;

			/******* buf 1 **/
			if(buf1Len > 0){
				log->_int.DORead.enable	   		= 1;
				log->_int.DORead.ident 	   		= log->_int.dwIdent;
				log->_int.DORead.pDestination 	= (UDINT) &buf1;
				log->_int.DORead.len		  	= buf1Len * log->_int.recLen;
				log->_int.DORead.Offset	   		= buf1Offset;

				/* Call FUB */
				if(log->_int.DOWrite.enable	== 0){;
					DatObjRead(&log->_int.DORead);
					log->_int.Status   = log->_int.DORead.status;
					if(log->_int.DORead.status == 0) log->_int.DORead.enable = 0;
					if(log->_int.Status == 20605){
						LoggerInit(log , log->_int.pLogID , log->_int.dbName , log->_int.MaxLogs);
						return 1;
					}
				}

				if(log->_int.DORead.enable == 0){
					for(i = (buf1Len -1) ; i >= 0  ; i--){
						if(k > (MAXLOGS -1)) break;

						p =  &buf1[i * log->_int.recLen];

						memcpy(&_dt , p , sizeof(plcdt));
						memcpy(&_t , p +  sizeof(plcdt), sizeof(plctime));

						SetTimeStamp(_t , _dt,&log->LogView[k] , &buf1[i * log->_int.recLen + sizeof(plcdt)+ sizeof(plcdt)]);

						k++;
					}
				}
				else return 0;
			}

			/******* buf 2 **/
			if(buf2Len > 0){
				log->_int.DORead.enable	   		= 1;
				log->_int.DORead.ident 	   		= log->_int.dwIdent;
				log->_int.DORead.pDestination 	= (UDINT) &buf2;
				log->_int.DORead.len		  	= buf2Len * log->_int.recLen;
				log->_int.DORead.Offset	   		= buf2Offset;

				/* Call FUB */
				if(log->_int.DOWrite.enable	== 0){;
					DatObjRead(&log->_int.DORead);
					log->_int.Status   = log->_int.DORead.status;
					if(log->_int.DORead.status == 0) log->_int.DORead.enable = 0;
					if(log->_int.Status == 20605){
						LoggerInit(log , log->_int.pLogID , log->_int.dbName , log->_int.MaxLogs);
						return 1;
					}
				}

				if(log->_int.DORead.enable == 0){
					for(i = (buf2Len -1) ; i >= 0  ; i--){
						if(k > (MAXLOGS -1)) break;

						p =  &buf2[i * log->_int.recLen];

						memcpy(&_dt , p , sizeof(plcdt));
						memcpy(&_t , p +  sizeof(plcdt), sizeof(plctime));

						SetTimeStamp(_t , _dt,&log->LogView[k] , &buf2[i * log->_int.recLen] + sizeof(plcdt)+ sizeof(plcdt));

						k++;
					}
				}
				else return 0;
			}

			log->Cmd.Refresh = 0;

		}
	}

	//int sprintf(char *out, const char *format, ...)

	int LogTxt(LOGMGR_obj *log , char *fmt, ...)
	{
	int ret ;
	char *pstr;
	va_list args;
	DTGetTime_typ DTGetTime_1;
	plcdt		_dt;
	plctime _t;
	char *where;
	int     retv;
  	va_list varg;

			if(!log->_int.DataObjReady) return -100;
			if(log->Cmd.PauseLog) 		return 102;

			where  = log->Logtxt_inp;
			va_start(varg, fmt);
			retv = xprint(xputs, &where, fmt, varg);
			*where = 0;
			va_end(varg);

			if(strlen(log->Logtxt_inp) >= MAXLOGINPUT)
				log->Logtxt_inp[MAXLOGINPUT-1] = 0;

			pstr = LEFT(log->Logtxt_inp , (strlen(log->Logtxt_inp) - 0));

			/* Get Date Time String */
			DTGetTime_1.enable = 1;
			DTGetTime(&DTGetTime_1);

			memset(log->_int.logBuf , 0 ,sizeof(log->_int.logBuf));
			memcpy(log->_int.logBuf , &DTGetTime_1.DT1 , sizeof(plcdt));
			_t = clock_ms();
			memcpy(log->_int.logBuf + sizeof(plcdt) ,&_t , sizeof(plctime));

			/*
			if(strlen(pstr)< MAXLOGINPUT){
				xsprintf((log->_int.logBuf + 8),"%s",pstr );

			}
			else{
				strcpy(log->_int.logBuf +  sizeof(plcdt) +  sizeof(plctime) , "log txt too long ");
			}
			*/

			xsprintf((log->_int.logBuf + 8),"%s",pstr );

			log->_int.DOWrite.enable	= 1;
		   	log->_int.DOWrite.ident		= log->_int.dwIdent;
		   	log->_int.DOWrite.Offset	= (*log->_int.pLogID) * log->_int.recLen;
		   	log->_int.DOWrite.pSource	= (UDINT)log->_int.logBuf ;
		   	log->_int.DOWrite.len		= log->_int.recLen;

		   	/* Call FUB */
			TRY_AGAIN:
		    DatObjWrite(&log->_int.DOWrite);
		   	log->_int.Status   = log->_int.DOWrite.status;

			if (log->_int.Status != 0 && log->_int.Status != 0xFFFF) // Error
				return -1;

			if(log->_int.Status == 0){
				(*log->_int.pLogID) ++;
				SetTimeStamp(_t , DTGetTime_1.DT1,log->LastLog , pstr);

			}
			else
				goto TRY_AGAIN;

			if((*log->_int.pLogID)> (log->_int.MaxLogs-1)) (*log->_int.pLogID) = 0;
				log->_int.DOWrite.enable	= 0;

			if(!log->Cmd.PauseRefreshNewLog)log->Cmd.Refresh = 1;

	        return ret;
	}

void SetTimeStamp(plctime t , plcdt dt, char * p , char * txt){

DTStructure _DTStruct;
TIMEStructure TimeStruct;

	DT_TO_DTStructure(dt, &_DTStruct);
	TIME_TO_TIMEStructure(t, (UDINT) &TimeStruct);
	//xsprintf(p,"%d-%02d:%02d:%02d-%d >%s" ,_DTStruct.day ,_DTStruct.hour , _DTStruct.minute , _DTStruct.second , TimeStruct.millisec , txt);
	//xsprintf(p,"%02d-%d >%s" , _DTStruct.second , TimeStruct.millisec , txt);
	xsprintf(p,"%02d:%02d:%02d-%d >%s" ,_DTStruct.hour , _DTStruct.minute , _DTStruct.second ,TimeStruct.millisec , txt);

	return;

}

DINT StreamToHex(USINT* inp , USINT* out , UINT num){
UINT i ;

	if(num == 0)
		return;

	for( i = 0; i < num ; i++){

		 strcpy(&out[i*3] , xultoa((UDINT)inp[i] , 16, 1));
		 out[i*3 + 2] = ' ';
	}
	out[i*3] = 0;

	return 1;

}

#endif
```

### LoggerLib.h
```c
/********************************************************************
 * COPYRIGHT -- PAI
 ********************************************************************
 * Library: Logger
 * File: LoggerLib.h
 * Author: Christopher
 * Created: December 26, 2008
 *******************************************************************/

#include <bur/plctypes.h>

//#include <..\bglib\bgsprintf.h>

#ifndef _LOGGERLIB_H
  	#define _LOGGERLIB_H

	#include <dataobj.h>
	#include <AsTime.h>
	#include <..\lib\xstring.c>

	#define MAXLOGS				20 // No of logs in View
	#define MAXLOGLEN			96 // Max log Len in View
	#define MAXLOGINPUT			48 // Log Rec len

	typedef struct LOGMGRCMD_obj
	{
		UINT scrollBy;
		plcbit ScrollUp;
		plcbit ScrollDwn;
		plcbit LastLogs;
		plcbit EnterLog;
		plcbit Refresh;
		plcbit PauseRefresh;
		plcbit PauseLog;
		plcbit PauseRefreshNewLog;
		plcbit EraseAllLogs;

	}LOGMGRCMD_obj;

	typedef struct LOGMGRINT_obj
	{
		UDINT *pLogID;
		plcbit DataObjReady;
		plcbit WriteData;
		plcbit ReadData;
		plcbit Create;
		unsigned short Status;
		UINT MaxLogs;
		char  logBuf[4+4+MAXLOGINPUT+1];
		plcstring  dbName[12+1];
		UDINT recLen;

		UDINT       		dwIdent;
		DatObjCreate_typ 	DOCreate;
		DatObjWrite_typ 	DOWrite;
		DatObjRead_typ  	DORead;
		DatObjInfo_typ  	DOInfo;

	}LOGMGRINT_obj;

	typedef struct LOGMGR_obj
	{
		plcstring LogView[MAXLOGS][MAXLOGLEN+1];
		plcstring LastLog[MAXLOGLEN+1];
		plcstring Logtxt_inp[128];
		plcbit	  Ready;
		UINT 	  curLog;
		LOGMGRINT_obj _int;
		LOGMGRCMD_obj Cmd;

	}LOGMGR_obj;

	/****************************************/
	/**    Functions Prototypes            **/

	DINT LoggerInit(LOGMGR_obj *log ,UDINT *Id, char *dbName , UINT maxLogs);
	DINT LoggerSrv(LOGMGR_obj *log);

	int LogTxt(LOGMGR_obj *log , char *fmt, ...);
	DINT StreamToHex(USINT* inp , USINT* out , UINT num);

	/****************************************/

#endif
```

### bgdebug.h
```c
#ifndef _BG_DEBUG_H
#define _BG_DEBUG_H

#include <..\Lib\utilityLib\bgsprintf.h>
#include <..\Lib\utilityLib\bgringbuffer.h>
#include <..\Lib\utilityLib\bgstring.h>
//Include required .c library files here. That way it's not needed in AS.
#include <..\Lib\utilityLib\bgringbuffer.c>
#include <..\Lib\utilityLib\bgsprintf.c>
#include <..\Lib\utilityLib\bgstring.c>

//#define DBG_CK(format, args...) bgRingBuffPrintf(&gRingBuffer, format, ## args); //Telnet
//#define DBG_CK(format, args...)  xsprintf(WarnTxt , format, ## args);   ERRxwarning(0xC350, 0, WarnTxt); // Logger in AS
//#define DBG_LogMgr(format, args...)  xsprintf(WarnTxt , format, ## args);   LogTxt(&LogMgr, WarnTxt); // LogBook on Pendant

#define DBG_CK(format, args...) ;
#define DBG_LogMgr(format, args...)  ;

#ifdef WIN32
#define DBG printf
#define DBGMSG printf

#define DBGCRT printf
#define DBGERR printf
#define DBGWAR printf
#define DBGINF printf
#define DBGDBG printf

#else

#include <bur/plc.h>
//#include "bgsprintf.h"
//#include "bgringbuffer.h"

#define BG_DEBUG_LEVEL_CRITICAL		0
#define BG_DEBUG_LEVEL_ERROR		1
#define BG_DEBUG_LEVEL_WARNING		2
#define BG_DEBUG_LEVEL_INFO			3
#define BG_DEBUG_LEVEL_DEBUG		4

#define BG_DEBUG_UNUSED	0x0

/*
- To completly remove debug msgs from the source code use:
#define BG_DEBUG_ENABLE 0
*/
#define BG_DEBUG_ENABLE 1

/*ptr to global ring buffer for debug messages*/
_GLOBAL bgRingBuffer_typ gRingBuffer;

#if BG_DEBUG_ENABLE == 1

//BG_DEBUG_ENABLE == 1 => debug messages present in the source code
#define DBG_OB(format, args...)  bgRingBuffPrintf(&gRingBuffer, format, ## args);
#define DBG(format, args...)  ;

//#define DBG(format, args...)	bgRingBuffPutDbgInfo(&gRingBuffer, __FILE__, __FUNCTION__, BG_DEBUG_LEVEL_CRITICAL, BG_DEBUG_UNUSED, format, ## args);
#define DBGMSG(format, args...)	bgRingBuffPrintf(&gRingBuffer, format, ## args);

#define DBGCRT(format, args...)	bgRingBuffPutDbgInfo(&gRingBuffer, __FILE__, __FUNCTION__, BG_DEBUG_LEVEL_CRITICAL, BG_DEBUG_UNUSED, format, ## args);
#define DBGERR(format, args...)	bgRingBuffPutDbgInfo(&gRingBuffer, __FILE__, __FUNCTION__, BG_DEBUG_LEVEL_ERROR, BG_DEBUG_UNUSED, format, ## args);
#define DBGWAR(format, args...)	bgRingBuffPutDbgInfo(&gRingBuffer, __FILE__, __FUNCTION__, BG_DEBUG_LEVEL_WARNING, BG_DEBUG_UNUSED, format, ## args);
#define DBGINF(format, args...)	bgRingBuffPutDbgInfo(&gRingBuffer, __FILE__, __FUNCTION__, BG_DEBUG_LEVEL_INFO, BG_DEBUG_UNUSED, format, ## args);
#define DBGDBG(format, args...)	bgRingBuffPutDbgInfo(&gRingBuffer, __FILE__, __FUNCTION__, BG_DEBUG_LEVEL_DEBUG, BG_DEBUG_UNUSED, format, ## args);

#else
/*BG_DEBUG_ENABLE == 0 => all debug messages removed from the source code*/

#define DBG_OB(format, args...)  	{};

#define DBG(format, args...)  		{};
#define DBGMSG(format, args...)  	{};

#define DBGCRT(format, args...)		{};
#define DBGERR(format, args...)		{};
#define DBGWAR(format, args...)		{};
#define DBGINF(format, args...)		{};
#define DBGDBG(format, args...)		{};

#endif /*#if BG_DEBUG_ENABLE*/

#endif /*#ifdef WIN32*/

#endif /*#ifndef _BG_DEBUG_H*/
```

### Handler.h - Attribute Definitions
```c
#ifndef _HANDLER_H
#define _HANDLER_H

#include <bur/plctypes.h>

#include <runtime.h>

_GLOBAL static UINT SEQUENCE_NUMBER;

/* Function Prototypes */
void handleArcLinkResponse ( Arc_Link_typ *arc);
void handleArcLinkRequests( Arc_Link_typ *arc);
void handleMasterToSlavesRequest( Arc_Link_typ *arc);
void handleMasterToSlaveRequest( Arc_Link_typ *arc);
void handlePeerToPeerRequest( Arc_Link_typ *arc);
void handlePeerToPeersRequest( Arc_Link_typ *arc);

/* Network Services */
void handleNetworkAction( Arc_Link_typ *arc);

/* Network Actions */
void processRecognitionActionArcLinkRequest( Arc_Link_typ *arc);
void processRecognitionActionArcLinkResponse( Arc_Link_typ *arc);
void processAssignNetworkAddressAction( Arc_Link_typ *arc);
void processAddToGroupAddressAction(Arc_Link_typ *arc); /* Action 5 */
void processGroupDataAction(Arc_Link_typ *arc); /* Action 2, Process Group Data Action */
void processNOP_ACTION(Arc_Link_typ *arc); /* Action 19 */
void processGetConfigurationObjectControlsAction(Arc_Link_typ *arc); /* Action 32 */
void processCreateEventReportAction(Arc_Link_typ *arc); /* Action 11*/
void processAttributeSearchAction(Arc_Link_typ *arc); /* Action 8 */

/* Network Blocks */
void handleNetworkBlock(Arc_Link_typ *arc);

/* Network block 0*/
void processReadNetworkConfigurationDataBlock(Arc_Link_typ *arc);
/* Read Network Configuration Data Response acknowledge */
void processReadNetworkConfigurationDataBlockResponse(Arc_Link_typ *arc);

/* Read Attributes */
void handleReadAttributeClassProperty(Arc_Link_typ *arc);
void handleReadAttributeValue(Arc_Link_typ *arc);

/* Write Atributes */
void handleWriteAttributeClassProperty(Arc_Link_typ *arc);
void handleWriteAttributeValue(Arc_Link_typ *arc);

/* handle unconfirmed Event Blocks, E.g. used with Telemetry */
void handleUnconfirmedEventBlock(Arc_Link_typ *arc);
void processTelemetryEvent(Arc_Link_typ *arc);
void processEnergyFBEvent(Arc_Link_typ *arc);
void processBlockMeterEvent(Arc_Link_typ *arc);
void processWeldScoreEvent(Arc_Link_typ *arc);

/* handle unconfirmed Event, E.g. arc change status*/
void handleUnconfirmedEvent(Arc_Link_typ *arc);
void processArcChangeStatusEvent(Arc_Link_typ *arc);

/* Key Methods */
void sendSuccesfullWriteAttributeConfirmation( Arc_Link_typ *arc);

/* write Message to Outgoing RingBuffer */
void writeMessageToOutgoingRingBuffer( Arc_Link_typ *arc);

/* Perform Misc Setup required for Telemetry */
void performRobotMiscSetup(Arc_Link_typ *arc);
void miscSetup(Arc_Link_typ *arc);
void createEventReport(Arc_Link_typ *arc);

/* Robot specific Commands */
void writeOutputOnCommand(Arc_Link_typ *arc);
void writeOutputOffCommand(Arc_Link_typ *arc);

void writeOutputCoolerOnCommand(Arc_Link_typ *arc);
void writeOutputCoolerOffCommand(Arc_Link_typ *arc);

void writeOutputGasEnableCommand(Arc_Link_typ *arc);
void writeOutputGasOnCommand(Arc_Link_typ *arc);
void writeOutputGasOffCommand(Arc_Link_typ *arc);

void createSetControlsAction(Arc_Link_typ *arc);
/* Create Weld Table Action To be tested */
void createWeldTableAction(Arc_Link_typ *arc);

//arc status change event
void processArcStatusChangeEvent(Arc_Link_typ *arc);

// process ready, faults status
void processStatusEvent(Arc_Link_typ *arc);

/* Read Attribute 30731 */
void readAttribute30731(Arc_Link_typ *arc);

/* handle fault status response */
void handleResponseAttribute30731(Arc_Link_typ *arc);

void action_ConfigDataSearch(Arc_Link_typ *arc);
void action_ConfigDataSearch_GasSol(Arc_Link_typ *arc);

/* handle Config Data Search response -  cooler Address*/
void handleResponseConfigDataSearchAction(Arc_Link_typ *arc);
void handleResponseConfigDataSearchAction_GasSol(Arc_Link_typ *arc);

void handleResponseReadControlParamDataAction(Arc_Link_typ *arc);

void readAttribute_CoolerSens(Arc_Link_typ *arc);
void handleResponse_ReadCoolerSens(Arc_Link_typ *arc);

void createReadCntrlParamDataAction(Arc_Link_typ *arc);

/*
	Error Logger by Obed Rev 1.0
*/
void log_error(Log_typ* err, char* msg);

#endif /* _HANDLER_H */
```
